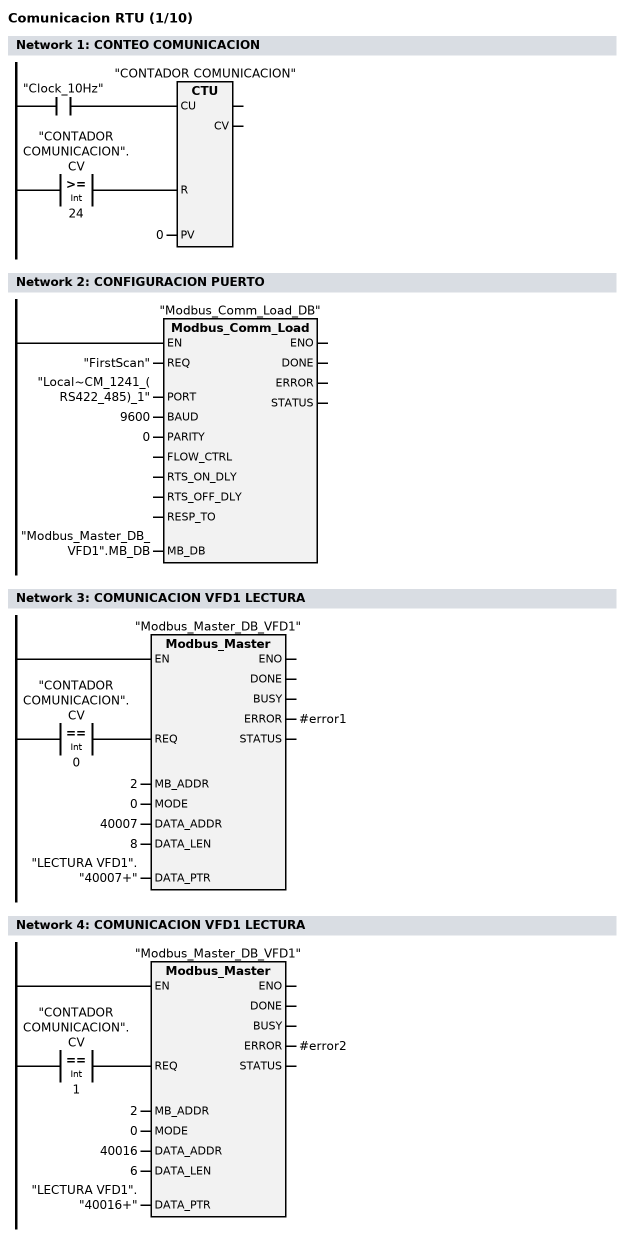
   "CONTADOR COMUNICACION".CTU(CU := "Clock_10Hz", R := "CONTADOR COMUNICACION".CV >= 24, PV := 0);
END_REGION

REGION Network 2: CONFIGURACION PUERTO
   "Modbus_Comm_Load_DB"(REQ := "FirstScan",   // Modbus_Comm_Load
                         PORT := "Local~CM_1241_(RS422_485)_1",
                         BAUD := 9600,
                         PARITY := 0,
                         MB_DB := "Modbus_Master_DB_VFD1".MB_DB);
END_REGION

REGION Network 3: COMUNICACION VFD1 LECTURA
   "Modbus_Master_DB_VFD1"(REQ := "CONTADOR COMUNICACION".CV = 0,   // Modbus_Master
                           MB_ADDR := 2,
                           MODE := 0,
                           DATA_ADDR := 40007,
                           DATA_LEN := 8,
                           DATA_PTR := "LECTURA VFD1"."40007+",
                           ERROR => #error1);
END_REGION

REGION Network 4: COMUNICACION VFD1 LECTURA
   "Modbus_Master_DB_VFD1"(REQ := "CONTADOR COMUNICACION".CV = 1,   // Modbus_Master
                           MB_ADDR := 2,
                           MODE := 0,
                           DATA_ADDR := 40016,
                           DATA_LEN := 6,
                           DATA_PTR := "LECTURA VFD1"."40016+",
                           ERROR => #error2);
END_REGION

REGION Network 5: COMUNICACION VFD2 LECTURA
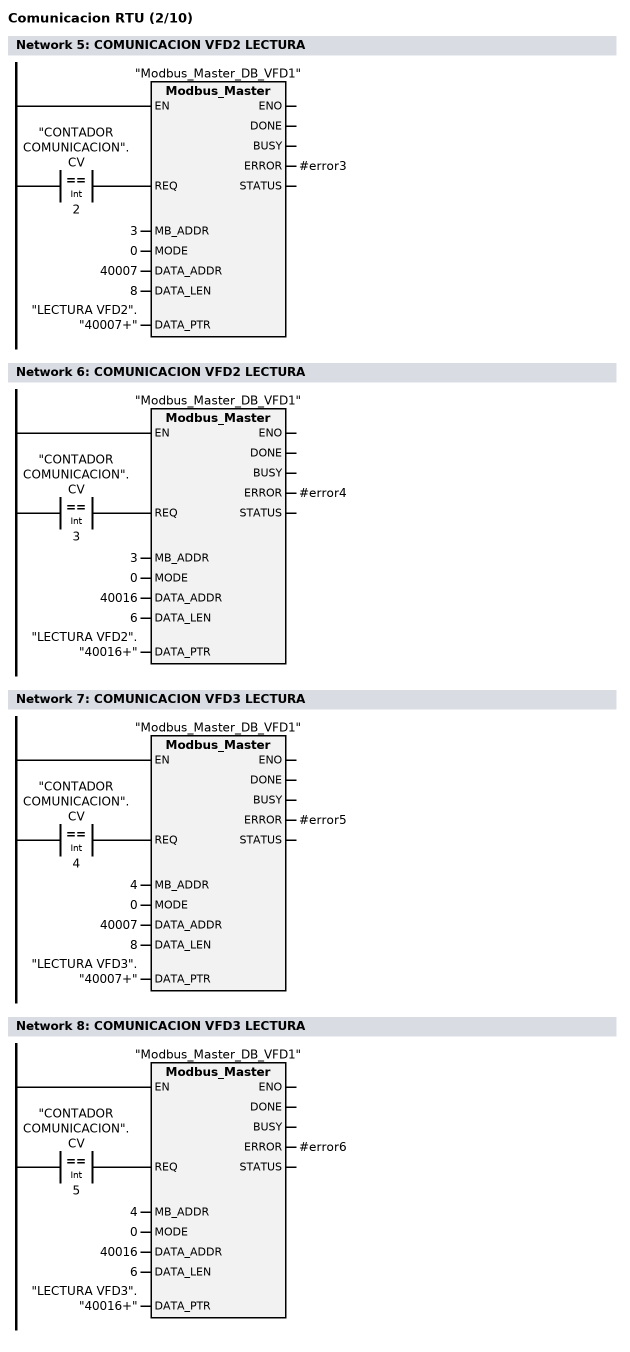
   "Modbus_Master_DB_VFD1"(REQ := "CONTADOR COMUNICACION".CV = 2,   // Modbus_Master
                           MB_ADDR := 3,
                           MODE := 0,
                           DATA_ADDR := 40007,
                           DATA_LEN := 8,
                           DATA_PTR := "LECTURA VFD2"."40007+",
                           ERROR => #error3);
END_REGION

REGION Network 6: COMUNICACION VFD2 LECTURA
   "Modbus_Master_DB_VFD1"(REQ := "CONTADOR COMUNICACION".CV = 3,   // Modbus_Master
                           MB_ADDR := 3,
                           MODE := 0,
                           DATA_ADDR := 40016,
                           DATA_LEN := 6,
                           DATA_PTR := "LECTURA VFD2"."40016+",
                           ERROR => #error4);
END_REGION

REGION Network 7: COMUNICACION VFD3 LECTURA
   "Modbus_Master_DB_VFD1"(REQ := "CONTADOR COMUNICACION".CV = 4,   // Modbus_Master
                           MB_ADDR := 4,
                           MODE := 0,
                           DATA_ADDR := 40007,
                           DATA_LEN := 8,
                           DATA_PTR := "LECTURA VFD3"."40007+",
                           ERROR => #error5);
END_REGION

REGION Network 8: COMUNICACION VFD3 LECTURA
   "Modbus_Master_DB_VFD1"(REQ := "CONTADOR COMUNICACION".CV = 5,   // Modbus_Master
                           MB_ADDR := 4,
                           MODE := 0,
                           DATA_ADDR := 40016,
                           DATA_LEN := 6,
                           DATA_PTR := "LECTURA VFD3"."40016+",
                           ERROR => #error6);
END_REGION

REGION Network 9: COMUNICACION VFD4 LECTURA
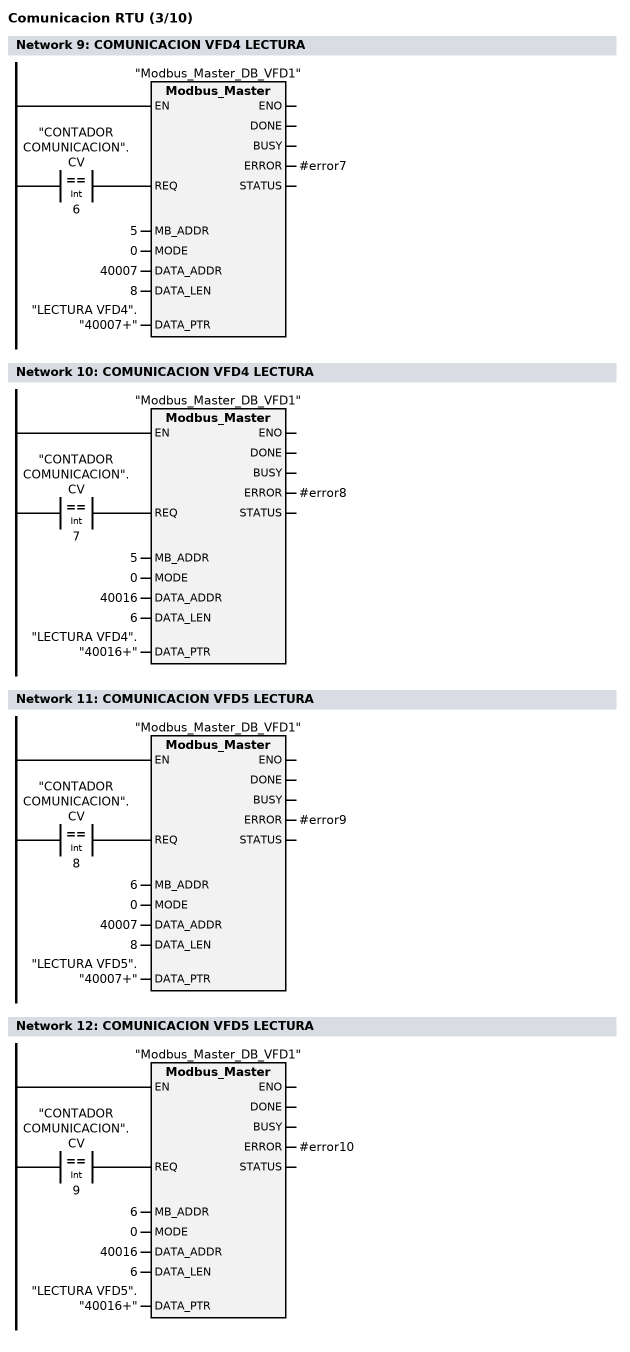
   "Modbus_Master_DB_VFD1"(REQ := "CONTADOR COMUNICACION".CV = 6,   // Modbus_Master
                           MB_ADDR := 5,
                           MODE := 0,
                           DATA_ADDR := 40007,
                           DATA_LEN := 8,
                           DATA_PTR := "LECTURA VFD4"."40007+",
                           ERROR => #error7);
END_REGION

REGION Network 10: COMUNICACION VFD4 LECTURA
   "Modbus_Master_DB_VFD1"(REQ := "CONTADOR COMUNICACION".CV = 7,   // Modbus_Master
                           MB_ADDR := 5,
                           MODE := 0,
                           DATA_ADDR := 40016,
                           DATA_LEN := 6,
                           DATA_PTR := "LECTURA VFD4"."40016+",
                           ERROR => #error8);
END_REGION

REGION Network 11: COMUNICACION VFD5 LECTURA
   "Modbus_Master_DB_VFD1"(REQ := "CONTADOR COMUNICACION".CV = 8,   // Modbus_Master
                           MB_ADDR := 6,
                           MODE := 0,
                           DATA_ADDR := 40007,
                           DATA_LEN := 8,
                           DATA_PTR := "LECTURA VFD5"."40007+",
                           ERROR => #error9);
END_REGION

REGION Network 12: COMUNICACION VFD5 LECTURA
   "Modbus_Master_DB_VFD1"(REQ := "CONTADOR COMUNICACION".CV = 9,   // Modbus_Master
                           MB_ADDR := 6,
                           MODE := 0,
                           DATA_ADDR := 40016,
                           DATA_LEN := 6,
                           DATA_PTR := "LECTURA VFD5"."40016+",
                           ERROR => #error10);
END_REGION

REGION Network 13: COMUNICACION VFD6 LECTURA
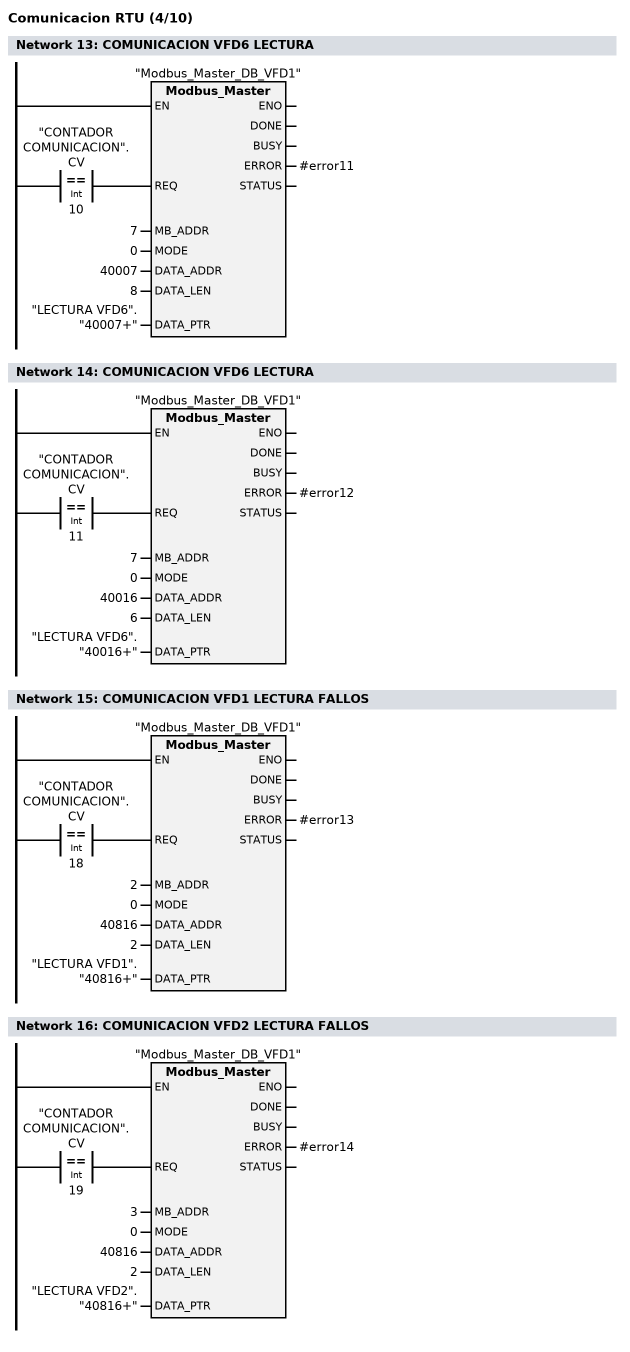
   "Modbus_Master_DB_VFD1"(REQ := "CONTADOR COMUNICACION".CV = 10,   // Modbus_Master
                           MB_ADDR := 7,
                           MODE := 0,
                           DATA_ADDR := 40007,
                           DATA_LEN := 8,
                           DATA_PTR := "LECTURA VFD6"."40007+",
                           ERROR => #error11);
END_REGION

REGION Network 14: COMUNICACION VFD6 LECTURA
   "Modbus_Master_DB_VFD1"(REQ := "CONTADOR COMUNICACION".CV = 11,   // Modbus_Master
                           MB_ADDR := 7,
                           MODE := 0,
                           DATA_ADDR := 40016,
                           DATA_LEN := 6,
                           DATA_PTR := "LECTURA VFD6"."40016+",
                           ERROR => #error12);
END_REGION

REGION Network 15: COMUNICACION VFD1 LECTURA FALLOS
   "Modbus_Master_DB_VFD1"(REQ := "CONTADOR COMUNICACION".CV = 18,   // Modbus_Master
                           MB_ADDR := 2,
                           MODE := 0,
                           DATA_ADDR := 40816,
                           DATA_LEN := 2,
                           DATA_PTR := "LECTURA VFD1"."40816+",
                           ERROR => #error13);
END_REGION

REGION Network 16: COMUNICACION VFD2 LECTURA FALLOS
   "Modbus_Master_DB_VFD1"(REQ := "CONTADOR COMUNICACION".CV = 19,   // Modbus_Master
                           MB_ADDR := 3,
                           MODE := 0,
                           DATA_ADDR := 40816,
                           DATA_LEN := 2,
                           DATA_PTR := "LECTURA VFD2"."40816+",
                           ERROR => #error14);
END_REGION

REGION Network 17: COMUNICACION VFD3 LECTURA FALLOS
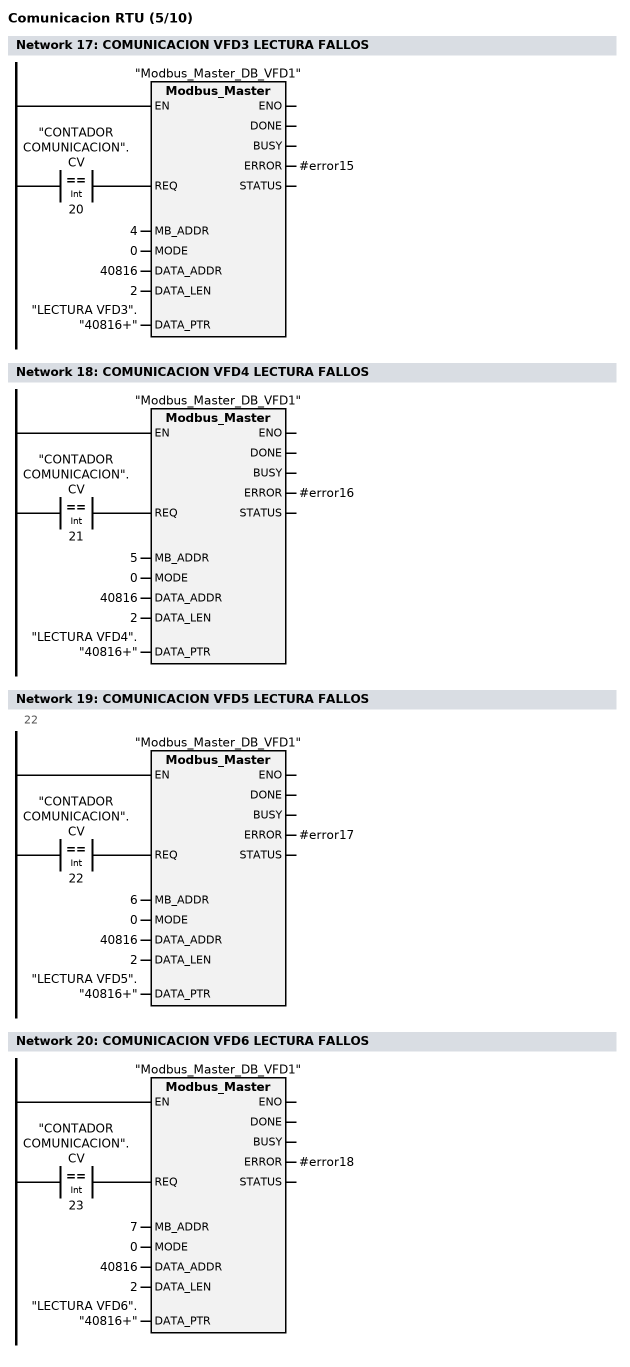
   "Modbus_Master_DB_VFD1"(REQ := "CONTADOR COMUNICACION".CV = 20,   // Modbus_Master
                           MB_ADDR := 4,
                           MODE := 0,
                           DATA_ADDR := 40816,
                           DATA_LEN := 2,
                           DATA_PTR := "LECTURA VFD3"."40816+",
                           ERROR => #error15);
END_REGION

REGION Network 18: COMUNICACION VFD4 LECTURA FALLOS
   "Modbus_Master_DB_VFD1"(REQ := "CONTADOR COMUNICACION".CV = 21,   // Modbus_Master
                           MB_ADDR := 5,
                           MODE := 0,
                           DATA_ADDR := 40816,
                           DATA_LEN := 2,
                           DATA_PTR := "LECTURA VFD4"."40816+",
                           ERROR => #error16);
END_REGION

REGION Network 19: COMUNICACION VFD5 LECTURA FALLOS
   // 22
   "Modbus_Master_DB_VFD1"(REQ := "CONTADOR COMUNICACION".CV = 22,   // Modbus_Master
                           MB_ADDR := 6,
                           MODE := 0,
                           DATA_ADDR := 40816,
                           DATA_LEN := 2,
                           DATA_PTR := "LECTURA VFD5"."40816+",
                           ERROR => #error17);
END_REGION

REGION Network 20: COMUNICACION VFD6 LECTURA FALLOS
   "Modbus_Master_DB_VFD1"(REQ := "CONTADOR COMUNICACION".CV = 23,   // Modbus_Master
                           MB_ADDR := 7,
                           MODE := 0,
                           DATA_ADDR := 40816,
                           DATA_LEN := 2,
                           DATA_PTR := "LECTURA VFD6"."40816+",
                           ERROR => #error18);
END_REGION

REGION Network 21: COMUNICACION VFD1 ESCRITURA
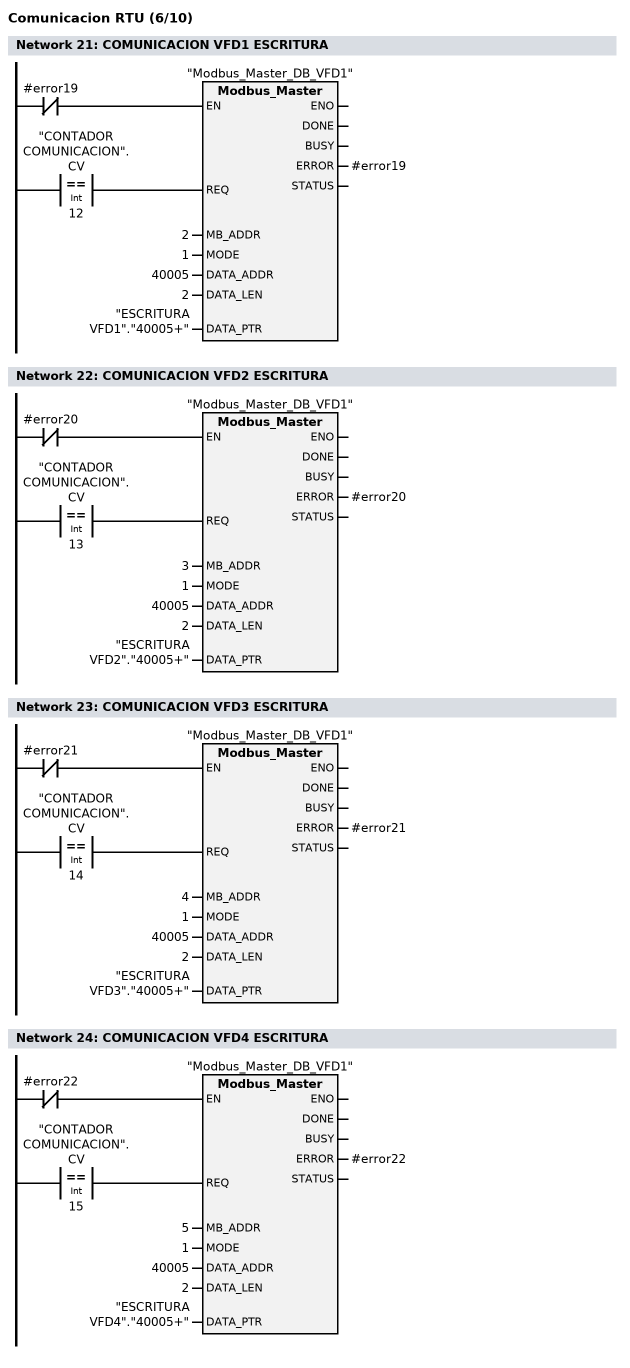
   IF NOT #error19 THEN
       "Modbus_Master_DB_VFD1"(REQ := "CONTADOR COMUNICACION".CV = 12,   // Modbus_Master
                               MB_ADDR := 2,
                               MODE := 1,
                               DATA_ADDR := 40005,
                               DATA_LEN := 2,
                               DATA_PTR := "ESCRITURA VFD1"."40005+",
                               ERROR => #error19);
   END_IF;
END_REGION

REGION Network 22: COMUNICACION VFD2 ESCRITURA
   IF NOT #error20 THEN
       "Modbus_Master_DB_VFD1"(REQ := "CONTADOR COMUNICACION".CV = 13,   // Modbus_Master
                               MB_ADDR := 3,
                               MODE := 1,
                               DATA_ADDR := 40005,
                               DATA_LEN := 2,
                               DATA_PTR := "ESCRITURA VFD2"."40005+",
                               ERROR => #error20);
   END_IF;
END_REGION

REGION Network 23: COMUNICACION VFD3 ESCRITURA
   IF NOT #error21 THEN
       "Modbus_Master_DB_VFD1"(REQ := "CONTADOR COMUNICACION".CV = 14,   // Modbus_Master
                               MB_ADDR := 4,
                               MODE := 1,
                               DATA_ADDR := 40005,
                               DATA_LEN := 2,
                               DATA_PTR := "ESCRITURA VFD3"."40005+",
                               ERROR => #error21);
   END_IF;
END_REGION

REGION Network 24: COMUNICACION VFD4 ESCRITURA
   IF NOT #error22 THEN
       "Modbus_Master_DB_VFD1"(REQ := "CONTADOR COMUNICACION".CV = 15,   // Modbus_Master
                               MB_ADDR := 5,
                               MODE := 1,
                               DATA_ADDR := 40005,
                               DATA_LEN := 2,
                               DATA_PTR := "ESCRITURA VFD4"."40005+",
                               ERROR => #error22);
   END_IF;
END_REGION

REGION Network 25: COMUNICACION VFD5 ESCRITURA
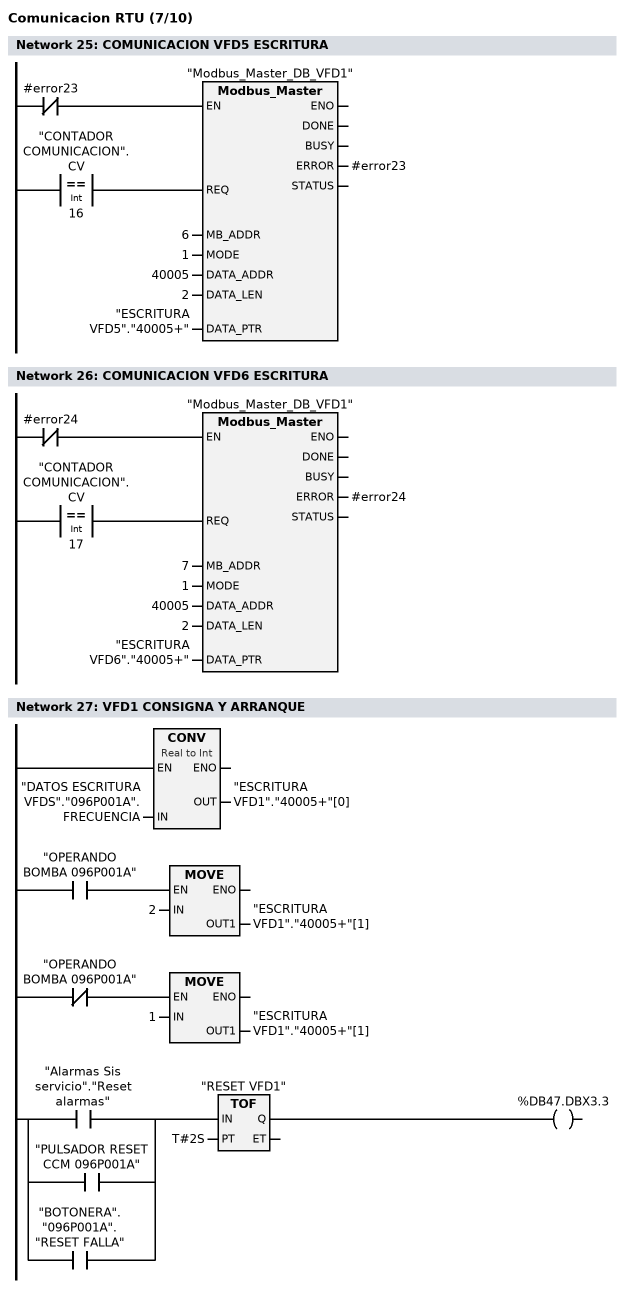
   IF NOT #error23 THEN
       "Modbus_Master_DB_VFD1"(REQ := "CONTADOR COMUNICACION".CV = 16,   // Modbus_Master
                               MB_ADDR := 6,
                               MODE := 1,
                               DATA_ADDR := 40005,
                               DATA_LEN := 2,
                               DATA_PTR := "ESCRITURA VFD5"."40005+",
                               ERROR => #error23);
   END_IF;
END_REGION

REGION Network 26: COMUNICACION VFD6 ESCRITURA
   IF NOT #error24 THEN
       "Modbus_Master_DB_VFD1"(REQ := "CONTADOR COMUNICACION".CV = 17,   // Modbus_Master
                               MB_ADDR := 7,
                               MODE := 1,
                               DATA_ADDR := 40005,
                               DATA_LEN := 2,
                               DATA_PTR := "ESCRITURA VFD6"."40005+",
                               ERROR => #error24);
   END_IF;
END_REGION

REGION Network 27: VFD1 CONSIGNA Y ARRANQUE
   "ESCRITURA VFD1"."40005+"[0] := REAL_TO_INT("DATOS ESCRITURA VFDS"."096P001A".FRECUENCIA);
   IF "OPERANDO BOMBA 096P001A" THEN "ESCRITURA VFD1"."40005+"[1] := 2; END_IF;
   IF NOT "OPERANDO BOMBA 096P001A" THEN "ESCRITURA VFD1"."40005+"[1] := 1; END_IF;
   "RESET VFD1".TOF(IN := "Alarmas Sis servicio"."Reset alarmas" OR "PULSADOR RESET CCM 096P001A" OR "BOTONERA"."096P001A"."RESET FALLA",
                    PT := T#2S);
   %DB47.DBX3.3 := "RESET VFD1".Q;
END_REGION

REGION Network 28: VFD2 CONSIGNA Y ARRANQUE
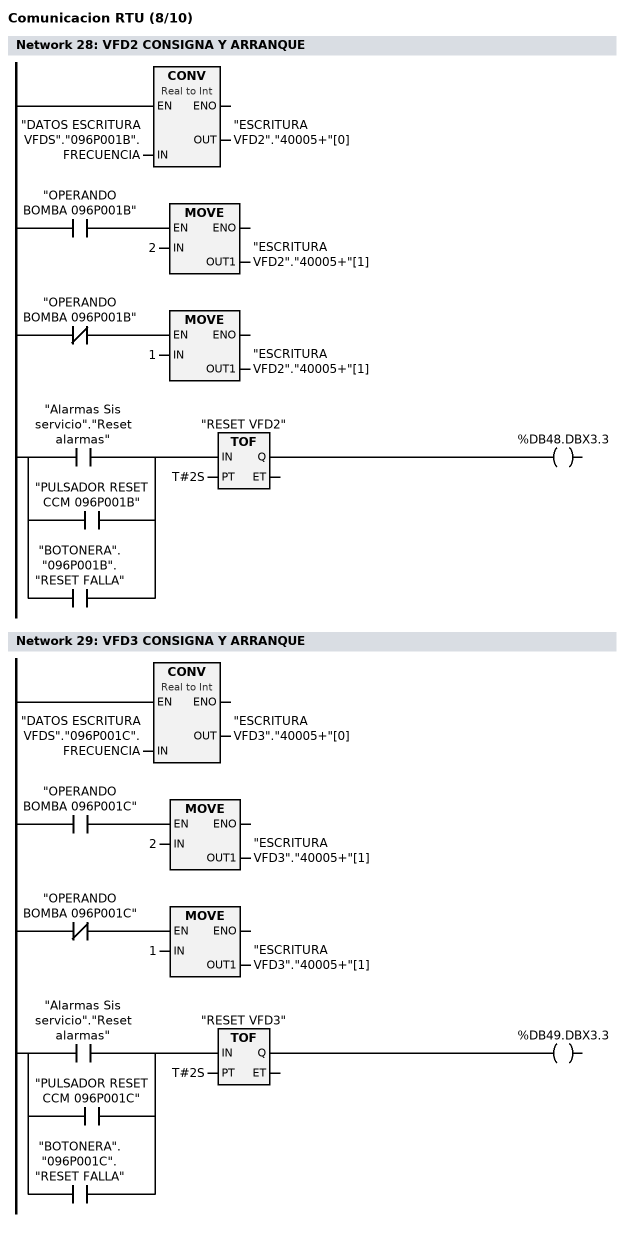
   "ESCRITURA VFD2"."40005+"[0] := REAL_TO_INT("DATOS ESCRITURA VFDS"."096P001B".FRECUENCIA);
   IF "OPERANDO BOMBA 096P001B" THEN "ESCRITURA VFD2"."40005+"[1] := 2; END_IF;
   IF NOT "OPERANDO BOMBA 096P001B" THEN "ESCRITURA VFD2"."40005+"[1] := 1; END_IF;
   "RESET VFD2".TOF(IN := "Alarmas Sis servicio"."Reset alarmas" OR "PULSADOR RESET CCM 096P001B" OR "BOTONERA"."096P001B"."RESET FALLA",
                    PT := T#2S);
   %DB48.DBX3.3 := "RESET VFD2".Q;
END_REGION

REGION Network 29: VFD3 CONSIGNA Y ARRANQUE
   "ESCRITURA VFD3"."40005+"[0] := REAL_TO_INT("DATOS ESCRITURA VFDS"."096P001C".FRECUENCIA);
   IF "OPERANDO BOMBA 096P001C" THEN "ESCRITURA VFD3"."40005+"[1] := 2; END_IF;
   IF NOT "OPERANDO BOMBA 096P001C" THEN "ESCRITURA VFD3"."40005+"[1] := 1; END_IF;
   "RESET VFD3".TOF(IN := "Alarmas Sis servicio"."Reset alarmas" OR "PULSADOR RESET CCM 096P001C" OR "BOTONERA"."096P001C"."RESET FALLA",
                    PT := T#2S);
   %DB49.DBX3.3 := "RESET VFD3".Q;
END_REGION

REGION Network 30: VFD4 CONSIGNA Y ARRANQUE
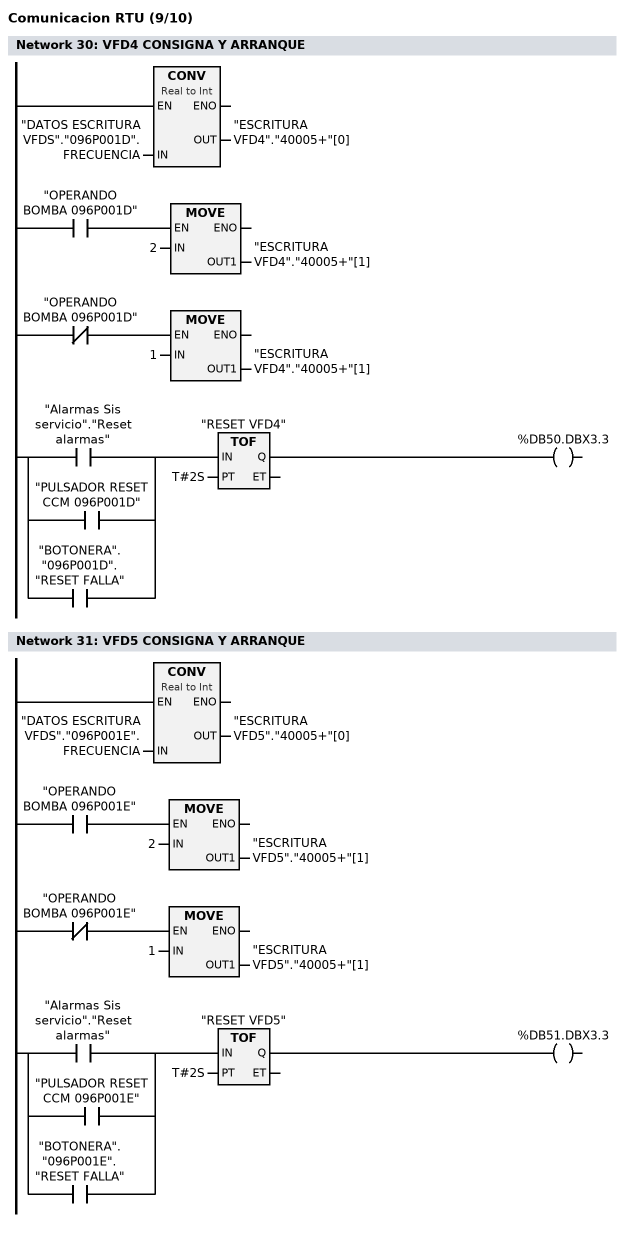
   "ESCRITURA VFD4"."40005+"[0] := REAL_TO_INT("DATOS ESCRITURA VFDS"."096P001D".FRECUENCIA);
   IF "OPERANDO BOMBA 096P001D" THEN "ESCRITURA VFD4"."40005+"[1] := 2; END_IF;
   IF NOT "OPERANDO BOMBA 096P001D" THEN "ESCRITURA VFD4"."40005+"[1] := 1; END_IF;
   "RESET VFD4".TOF(IN := "Alarmas Sis servicio"."Reset alarmas" OR "PULSADOR RESET CCM 096P001D" OR "BOTONERA"."096P001D"."RESET FALLA",
                    PT := T#2S);
   %DB50.DBX3.3 := "RESET VFD4".Q;
END_REGION

REGION Network 31: VFD5 CONSIGNA Y ARRANQUE
   "ESCRITURA VFD5"."40005+"[0] := REAL_TO_INT("DATOS ESCRITURA VFDS"."096P001E".FRECUENCIA);
   IF "OPERANDO BOMBA 096P001E" THEN "ESCRITURA VFD5"."40005+"[1] := 2; END_IF;
   IF NOT "OPERANDO BOMBA 096P001E" THEN "ESCRITURA VFD5"."40005+"[1] := 1; END_IF;
   "RESET VFD5".TOF(IN := "Alarmas Sis servicio"."Reset alarmas" OR "PULSADOR RESET CCM 096P001E" OR "BOTONERA"."096P001E"."RESET FALLA",
                    PT := T#2S);
   %DB51.DBX3.3 := "RESET VFD5".Q;
END_REGION

REGION Network 32: VFD6 CONSIGNA Y ARRANQUE
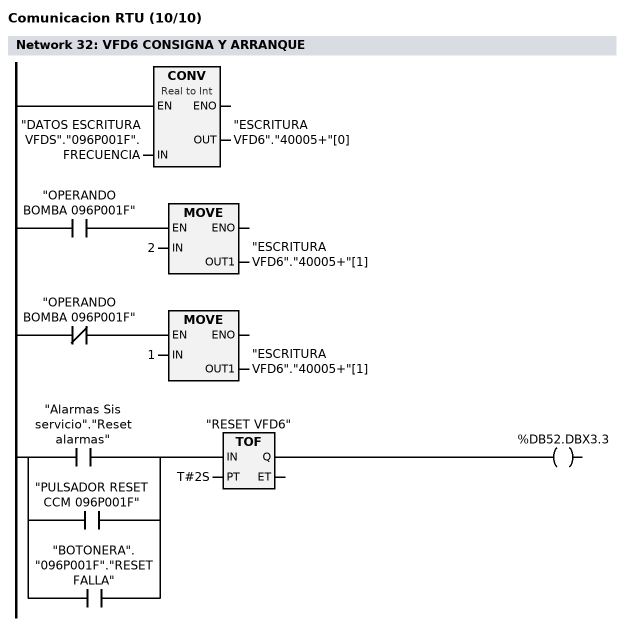
   "ESCRITURA VFD6"."40005+"[0] := REAL_TO_INT("DATOS ESCRITURA VFDS"."096P001F".FRECUENCIA);
   IF "OPERANDO BOMBA 096P001F" THEN "ESCRITURA VFD6"."40005+"[1] := 2; END_IF;
   IF NOT "OPERANDO BOMBA 096P001F" THEN "ESCRITURA VFD6"."40005+"[1] := 1; END_IF;
   "RESET VFD6".TOF(IN := "Alarmas Sis servicio"."Reset alarmas" OR "PULSADOR RESET CCM 096P001F" OR "BOTONERA"."096P001F"."RESET FALLA",
                    PT := T#2S);
   %DB52.DBX3.3 := "RESET VFD6".Q;
END_REGION
END_FUNCTION

FUNCTION "DATOS HMI" : Void   // FC6, LAD
{ S7_Optimized_Access := 'TRUE' }
VERSION : 0.1
BEGIN

REGION Network 1: VFD1
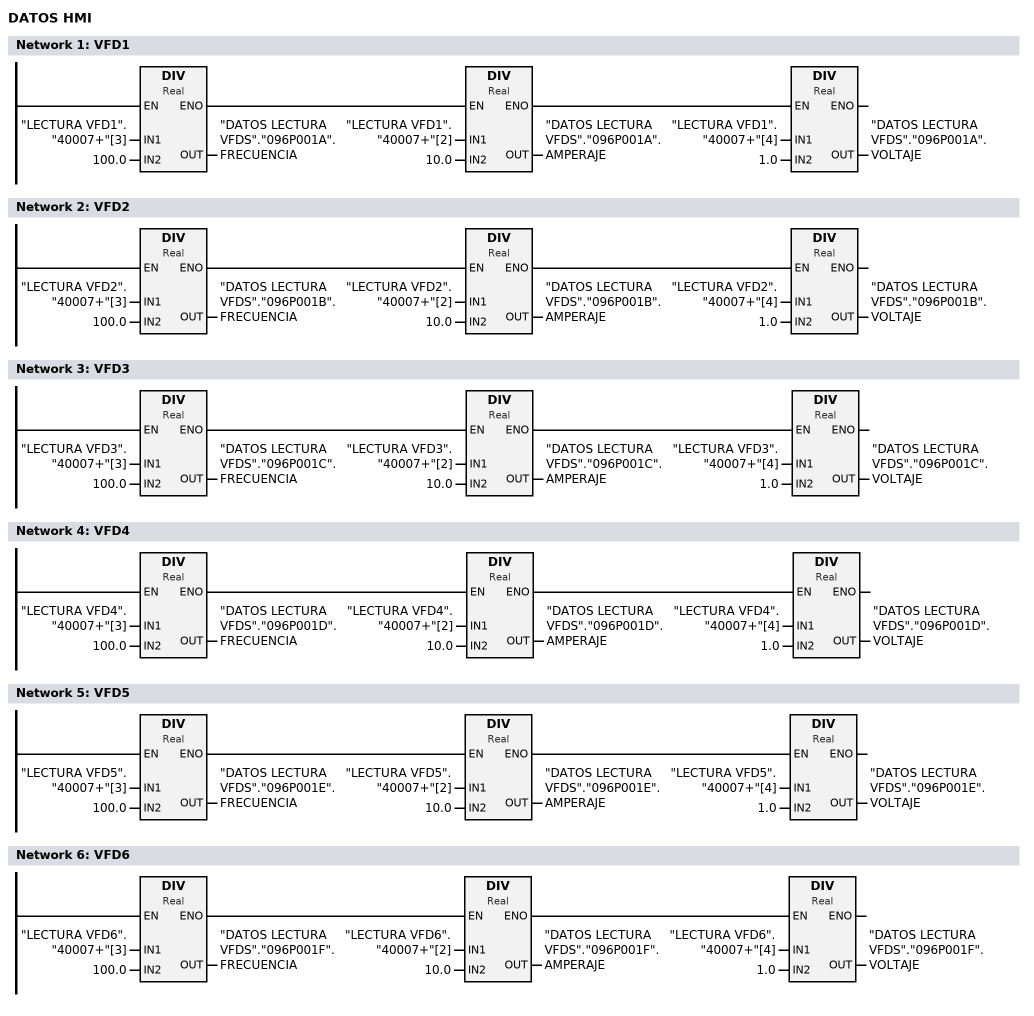
   RUNG wire#powerrail
      { S7_Templates := "SrcType := Real" } Div(in1 := "LECTURA VFD1"."40007+"[3], in2 := 100.0, out => "DATOS LECTURA VFDS"."096P001A".FRECUENCIA)
      { S7_Templates := "SrcType := Real" } Div(in1 := "LECTURA VFD1"."40007+"[2], in2 := 10.0, out => "DATOS LECTURA VFDS"."096P001A".AMPERAJE)
      { S7_Templates := "SrcType := Real" } Div(in1 := "LECTURA VFD1"."40007+"[4], in2 := 1.0, out => "DATOS LECTURA VFDS"."096P001A".VOLTAJE)
   END_RUNG
   // the same network as SCL:
   "DATOS LECTURA VFDS"."096P001A".FRECUENCIA := "LECTURA VFD1"."40007+"[3] / 100.0;
   "DATOS LECTURA VFDS"."096P001A".AMPERAJE := "LECTURA VFD1"."40007+"[2] / 10.0;
   "DATOS LECTURA VFDS"."096P001A".VOLTAJE := "LECTURA VFD1"."40007+"[4] / 1.0;
END_REGION

REGION Network 2: VFD2
   RUNG wire#powerrail
      { S7_Templates := "SrcType := Real" } Div(in1 := "LECTURA VFD2"."40007+"[3], in2 := 100.0, out => "DATOS LECTURA VFDS"."096P001B".FRECUENCIA)
      { S7_Templates := "SrcType := Real" } Div(in1 := "LECTURA VFD2"."40007+"[2], in2 := 10.0, out => "DATOS LECTURA VFDS"."096P001B".AMPERAJE)
      { S7_Templates := "SrcType := Real" } Div(in1 := "LECTURA VFD2"."40007+"[4], in2 := 1.0, out => "DATOS LECTURA VFDS"."096P001B".VOLTAJE)
   END_RUNG
   // the same network as SCL:
   "DATOS LECTURA VFDS"."096P001B".FRECUENCIA := "LECTURA VFD2"."40007+"[3] / 100.0;
   "DATOS LECTURA VFDS"."096P001B".AMPERAJE := "LECTURA VFD2"."40007+"[2] / 10.0;
   "DATOS LECTURA VFDS"."096P001B".VOLTAJE := "LECTURA VFD2"."40007+"[4] / 1.0;
END_REGION

REGION Network 3: VFD3
   RUNG wire#powerrail
      { S7_Templates := "SrcType := Real" } Div(in1 := "LECTURA VFD3"."40007+"[3], in2 := 100.0, out => "DATOS LECTURA VFDS"."096P001C".FRECUENCIA)
      { S7_Templates := "SrcType := Real" } Div(in1 := "LECTURA VFD3"."40007+"[2], in2 := 10.0, out => "DATOS LECTURA VFDS"."096P001C".AMPERAJE)
      { S7_Templates := "SrcType := Real" } Div(in1 := "LECTURA VFD3"."40007+"[4], in2 := 1.0, out => "DATOS LECTURA VFDS"."096P001C".VOLTAJE)
   END_RUNG
   // the same network as SCL:
   "DATOS LECTURA VFDS"."096P001C".FRECUENCIA := "LECTURA VFD3"."40007+"[3] / 100.0;
   "DATOS LECTURA VFDS"."096P001C".AMPERAJE := "LECTURA VFD3"."40007+"[2] / 10.0;
   "DATOS LECTURA VFDS"."096P001C".VOLTAJE := "LECTURA VFD3"."40007+"[4] / 1.0;
END_REGION

REGION Network 4: VFD4
   RUNG wire#powerrail
      { S7_Templates := "SrcType := Real" } Div(in1 := "LECTURA VFD4"."40007+"[3], in2 := 100.0, out => "DATOS LECTURA VFDS"."096P001D".FRECUENCIA)
      { S7_Templates := "SrcType := Real" } Div(in1 := "LECTURA VFD4"."40007+"[2], in2 := 10.0, out => "DATOS LECTURA VFDS"."096P001D".AMPERAJE)
      { S7_Templates := "SrcType := Real" } Div(in1 := "LECTURA VFD4"."40007+"[4], in2 := 1.0, out => "DATOS LECTURA VFDS"."096P001D".VOLTAJE)
   END_RUNG
   // the same network as SCL:
   "DATOS LECTURA VFDS"."096P001D".FRECUENCIA := "LECTURA VFD4"."40007+"[3] / 100.0;
   "DATOS LECTURA VFDS"."096P001D".AMPERAJE := "LECTURA VFD4"."40007+"[2] / 10.0;
   "DATOS LECTURA VFDS"."096P001D".VOLTAJE := "LECTURA VFD4"."40007+"[4] / 1.0;
END_REGION

REGION Network 5: VFD5
   RUNG wire#powerrail
      { S7_Templates := "SrcType := Real" } Div(in1 := "LECTURA VFD5"."40007+"[3], in2 := 100.0, out => "DATOS LECTURA VFDS"."096P001E".FRECUENCIA)
      { S7_Templates := "SrcType := Real" } Div(in1 := "LECTURA VFD5"."40007+"[2], in2 := 10.0, out => "DATOS LECTURA VFDS"."096P001E".AMPERAJE)
      { S7_Templates := "SrcType := Real" } Div(in1 := "LECTURA VFD5"."40007+"[4], in2 := 1.0, out => "DATOS LECTURA VFDS"."096P001E".VOLTAJE)
   END_RUNG
   // the same network as SCL:
   "DATOS LECTURA VFDS"."096P001E".FRECUENCIA := "LECTURA VFD5"."40007+"[3] / 100.0;
   "DATOS LECTURA VFDS"."096P001E".AMPERAJE := "LECTURA VFD5"."40007+"[2] / 10.0;
   "DATOS LECTURA VFDS"."096P001E".VOLTAJE := "LECTURA VFD5"."40007+"[4] / 1.0;
END_REGION

REGION Network 6: VFD6
   RUNG wire#powerrail
      { S7_Templates := "SrcType := Real" } Div(in1 := "LECTURA VFD6"."40007+"[3], in2 := 100.0, out => "DATOS LECTURA VFDS"."096P001F".FRECUENCIA)
      { S7_Templates := "SrcType := Real" } Div(in1 := "LECTURA VFD6"."40007+"[2], in2 := 10.0, out => "DATOS LECTURA VFDS"."096P001F".AMPERAJE)
      { S7_Templates := "SrcType := Real" } Div(in1 := "LECTURA VFD6"."40007+"[4], in2 := 1.0, out => "DATOS LECTURA VFDS"."096P001F".VOLTAJE)
   END_RUNG
   // the same network as SCL:
   "DATOS LECTURA VFDS"."096P001F".FRECUENCIA := "LECTURA VFD6"."40007+"[3] / 100.0;
   "DATOS LECTURA VFDS"."096P001F".AMPERAJE := "LECTURA VFD6"."40007+"[2] / 10.0;
   "DATOS LECTURA VFDS"."096P001F".VOLTAJE := "LECTURA VFD6"."40007+"[4] / 1.0;
END_REGION
END_FUNCTION

FUNCTION "COMUNICACION MODBUS TCP" : Void   // FC7, LAD
{ S7_Optimized_Access := 'TRUE' }
VERSION : 0.1
   VAR_TEMP
      "REAL 1" : Real;
      "REAL 2" : Real;
      "REAL 3" : Real;
      "REAL 4" : Real;
      "REAL 5" : Real;
      "REAL 6" : Real;
      "REAL 7" : Real;
      "REAL 8" : Real;
      "REAL 9" : Real;
      "REAL 10" : Real;
      "REAL 11" : Real;
      "REAL 12" : Real;
      "REAL 13" : Real;
      "REAL 14" : Real;
      "REAL 15" : Real;
      "REAL 16" : Real;
      "REAL 17" : Real;
      "REAL 18" : Real;
      "REAL 19" : Real;
      "REAL 20" : Real;
      "REAL 21" : Real;
      "REAL 22" : Real;
      "REAL 23" : Real;
      "REAL 24" : Real;
      "REAL 25" : Real;
      "REAL 26" : Real;
      "REAL 27" : Real;
      "REAL 28" : Real;
      "REAL 29" : Real;
      "REAL 30" : Real;
   END_VAR
   VAR_TEMP   // added for the SCL form of the ladder/FBD networks
      _w1 : Bool;
      _w2 : Bool;
      _w3 : Bool;
   END_VAR
BEGIN

REGION Network 1: CONFIGURACION MODBUS TCP
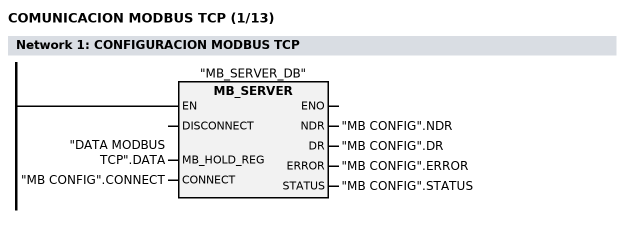
   "MB_SERVER_DB"(MB_HOLD_REG := "DATA MODBUS TCP".DATA,   // MB_SERVER
                  CONNECT := "MB CONFIG".CONNECT,
                  NDR => "MB CONFIG".NDR,
                  DR => "MB CONFIG".DR,
                  ERROR => "MB CONFIG".ERROR,
                  STATUS => "MB CONFIG".STATUS);
END_REGION

REGION Network 2: ENTRADAS DIGITALES
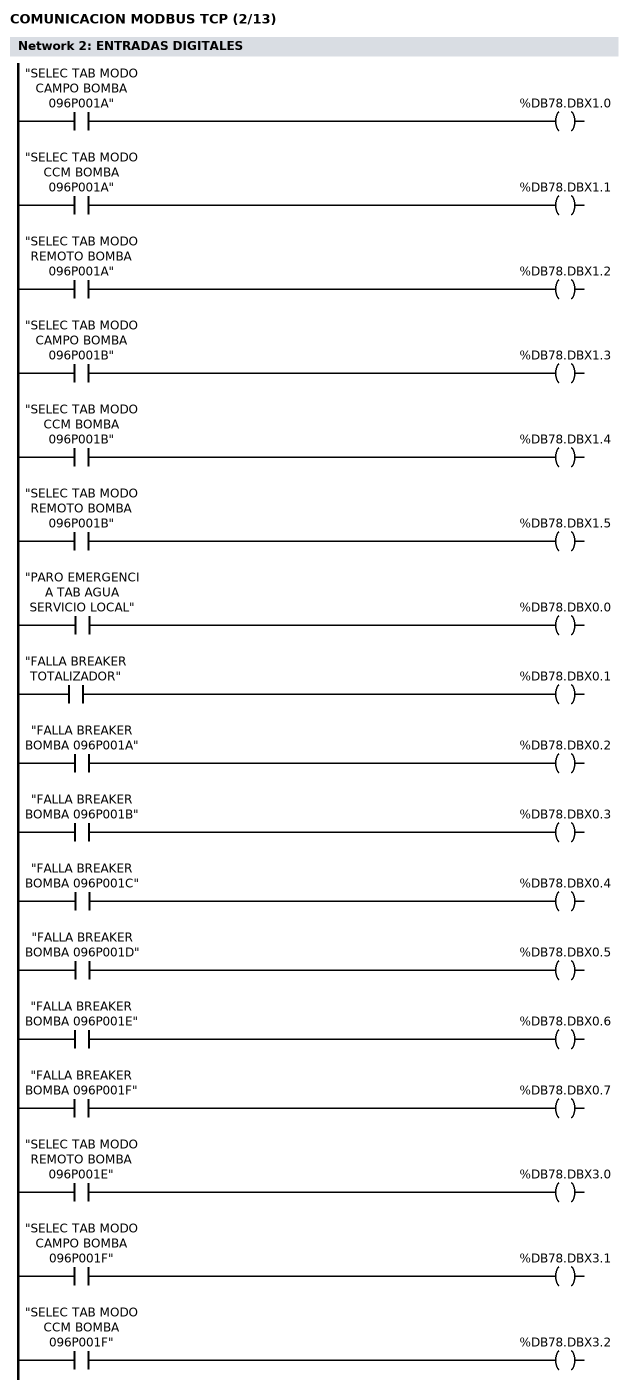
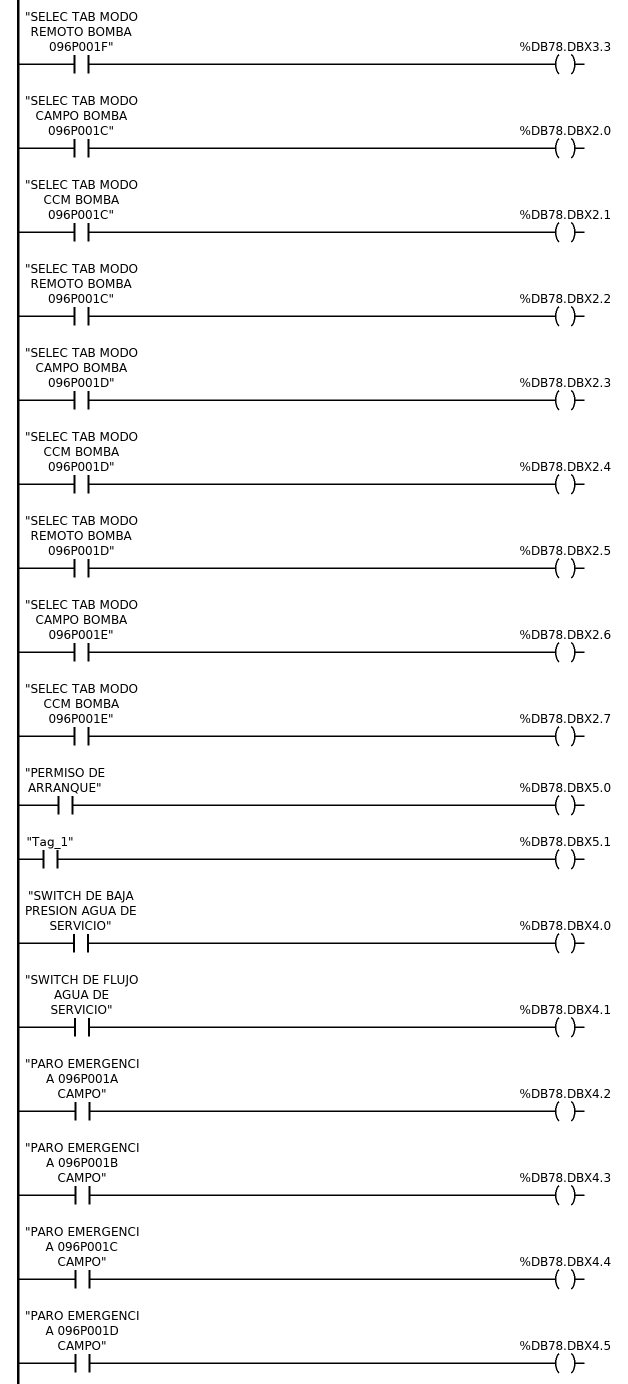
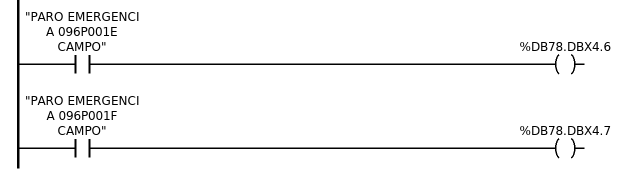
   RUNG wire#powerrail
      Contact( "SELEC TAB MODO CAMPO BOMBA 096P001A" )
      Coil( %DB78.DBX1.0 )
   END_RUNG
   RUNG wire#powerrail
      Contact( "SELEC TAB MODO CCM BOMBA 096P001A" )
      Coil( %DB78.DBX1.1 )
   END_RUNG
   RUNG wire#powerrail
      Contact( "SELEC TAB MODO REMOTO BOMBA 096P001A" )
      Coil( %DB78.DBX1.2 )
   END_RUNG
   RUNG wire#powerrail
      Contact( "SELEC TAB MODO CAMPO BOMBA 096P001B" )
      Coil( %DB78.DBX1.3 )
   END_RUNG
   RUNG wire#powerrail
      Contact( "SELEC TAB MODO CCM BOMBA 096P001B" )
      Coil( %DB78.DBX1.4 )
   END_RUNG
   RUNG wire#powerrail
      Contact( "SELEC TAB MODO REMOTO BOMBA 096P001B" )
      Coil( %DB78.DBX1.5 )
   END_RUNG
   RUNG wire#powerrail
      Contact( "PARO EMERGENCIA TAB AGUA SERVICIO LOCAL" )
      Coil( %DB78.DBX0.0 )
   END_RUNG
   RUNG wire#powerrail
      Contact( "FALLA BREAKER TOTALIZADOR" )
      Coil( %DB78.DBX0.1 )
   END_RUNG
   RUNG wire#powerrail
      Contact( "FALLA BREAKER BOMBA 096P001A" )
      Coil( %DB78.DBX0.2 )
   END_RUNG
   RUNG wire#powerrail
      Contact( "FALLA BREAKER BOMBA 096P001B" )
      Coil( %DB78.DBX0.3 )
   END_RUNG
   RUNG wire#powerrail
      Contact( "FALLA BREAKER BOMBA 096P001C" )
      Coil( %DB78.DBX0.4 )
   END_RUNG
   RUNG wire#powerrail
      Contact( "FALLA BREAKER BOMBA 096P001D" )
      Coil( %DB78.DBX0.5 )
   END_RUNG
   RUNG wire#powerrail
      Contact( "FALLA BREAKER BOMBA 096P001E" )
      Coil( %DB78.DBX0.6 )
   END_RUNG
   RUNG wire#powerrail
      Contact( "FALLA BREAKER BOMBA 096P001F" )
      Coil( %DB78.DBX0.7 )
   END_RUNG
   RUNG wire#powerrail
      Contact( "SELEC TAB MODO REMOTO BOMBA 096P001E" )
      Coil( %DB78.DBX3.0 )
   END_RUNG
   RUNG wire#powerrail
      Contact( "SELEC TAB MODO CAMPO BOMBA 096P001F" )
      Coil( %DB78.DBX3.1 )
   END_RUNG
   RUNG wire#powerrail
      Contact( "SELEC TAB MODO CCM BOMBA 096P001F" )
      Coil( %DB78.DBX3.2 )
   END_RUNG
   RUNG wire#powerrail
      Contact( "SELEC TAB MODO REMOTO BOMBA 096P001F" )
      Coil( %DB78.DBX3.3 )
   END_RUNG
   RUNG wire#powerrail
      Contact( "SELEC TAB MODO CAMPO BOMBA 096P001C" )
      Coil( %DB78.DBX2.0 )
   END_RUNG
   RUNG wire#powerrail
      Contact( "SELEC TAB MODO CCM BOMBA 096P001C" )
      Coil( %DB78.DBX2.1 )
   END_RUNG
   RUNG wire#powerrail
      Contact( "SELEC TAB MODO REMOTO BOMBA 096P001C" )
      Coil( %DB78.DBX2.2 )
   END_RUNG
   RUNG wire#powerrail
      Contact( "SELEC TAB MODO CAMPO BOMBA 096P001D" )
      Coil( %DB78.DBX2.3 )
   END_RUNG
   RUNG wire#powerrail
      Contact( "SELEC TAB MODO CCM BOMBA 096P001D" )
      Coil( %DB78.DBX2.4 )
   END_RUNG
   RUNG wire#powerrail
      Contact( "SELEC TAB MODO REMOTO BOMBA 096P001D" )
      Coil( %DB78.DBX2.5 )
   END_RUNG
   RUNG wire#powerrail
      Contact( "SELEC TAB MODO CAMPO BOMBA 096P001E" )
      Coil( %DB78.DBX2.6 )
   END_RUNG
   RUNG wire#powerrail
      Contact( "SELEC TAB MODO CCM BOMBA 096P001E" )
      Coil( %DB78.DBX2.7 )
   END_RUNG
   RUNG wire#powerrail
      Contact( "PERMISO DE ARRANQUE" )
      Coil( %DB78.DBX5.0 )
   END_RUNG
   RUNG wire#powerrail
      Contact( "Tag_1" )
      Coil( %DB78.DBX5.1 )
   END_RUNG
   RUNG wire#powerrail
      Contact( "SWITCH DE BAJA PRESION AGUA DE SERVICIO" )
      Coil( %DB78.DBX4.0 )
   END_RUNG
   RUNG wire#powerrail
      Contact( "SWITCH DE FLUJO AGUA DE SERVICIO" )
      Coil( %DB78.DBX4.1 )
   END_RUNG
   RUNG wire#powerrail
      Contact( "PARO EMERGENCIA 096P001A CAMPO" )
      Coil( %DB78.DBX4.2 )
   END_RUNG
   RUNG wire#powerrail
      Contact( "PARO EMERGENCIA 096P001B CAMPO" )
      Coil( %DB78.DBX4.3 )
   END_RUNG
   RUNG wire#powerrail
      Contact( "PARO EMERGENCIA 096P001C CAMPO" )
      Coil( %DB78.DBX4.4 )
   END_RUNG
   RUNG wire#powerrail
      Contact( "PARO EMERGENCIA 096P001D CAMPO" )
      Coil( %DB78.DBX4.5 )
   END_RUNG
   RUNG wire#powerrail
      Contact( "PARO EMERGENCIA 096P001E CAMPO" )
      Coil( %DB78.DBX4.6 )
   END_RUNG
   RUNG wire#powerrail
      Contact( "PARO EMERGENCIA 096P001F CAMPO" )
      Coil( %DB78.DBX4.7 )
   END_RUNG
   // the same network as SCL:
   %DB78.DBX1.0 := "SELEC TAB MODO CAMPO BOMBA 096P001A";
   %DB78.DBX1.1 := "SELEC TAB MODO CCM BOMBA 096P001A";
   %DB78.DBX1.2 := "SELEC TAB MODO REMOTO BOMBA 096P001A";
   %DB78.DBX1.3 := "SELEC TAB MODO CAMPO BOMBA 096P001B";
   %DB78.DBX1.4 := "SELEC TAB MODO CCM BOMBA 096P001B";
   %DB78.DBX1.5 := "SELEC TAB MODO REMOTO BOMBA 096P001B";
   %DB78.DBX0.0 := "PARO EMERGENCIA TAB AGUA SERVICIO LOCAL";
   %DB78.DBX0.1 := "FALLA BREAKER TOTALIZADOR";
   %DB78.DBX0.2 := "FALLA BREAKER BOMBA 096P001A";
   %DB78.DBX0.3 := "FALLA BREAKER BOMBA 096P001B";
   %DB78.DBX0.4 := "FALLA BREAKER BOMBA 096P001C";
   %DB78.DBX0.5 := "FALLA BREAKER BOMBA 096P001D";
   %DB78.DBX0.6 := "FALLA BREAKER BOMBA 096P001E";
   %DB78.DBX0.7 := "FALLA BREAKER BOMBA 096P001F";
   %DB78.DBX3.0 := "SELEC TAB MODO REMOTO BOMBA 096P001E";
   %DB78.DBX3.1 := "SELEC TAB MODO CAMPO BOMBA 096P001F";
   %DB78.DBX3.2 := "SELEC TAB MODO CCM BOMBA 096P001F";
   %DB78.DBX3.3 := "SELEC TAB MODO REMOTO BOMBA 096P001F";
   %DB78.DBX2.0 := "SELEC TAB MODO CAMPO BOMBA 096P001C";
   %DB78.DBX2.1 := "SELEC TAB MODO CCM BOMBA 096P001C";
   %DB78.DBX2.2 := "SELEC TAB MODO REMOTO BOMBA 096P001C";
   %DB78.DBX2.3 := "SELEC TAB MODO CAMPO BOMBA 096P001D";
   %DB78.DBX2.4 := "SELEC TAB MODO CCM BOMBA 096P001D";
   %DB78.DBX2.5 := "SELEC TAB MODO REMOTO BOMBA 096P001D";
   %DB78.DBX2.6 := "SELEC TAB MODO CAMPO BOMBA 096P001E";
   %DB78.DBX2.7 := "SELEC TAB MODO CCM BOMBA 096P001E";
   %DB78.DBX5.0 := "PERMISO DE ARRANQUE";
   %DB78.DBX5.1 := "Tag_1";
   %DB78.DBX4.0 := "SWITCH DE BAJA PRESION AGUA DE SERVICIO";
   %DB78.DBX4.1 := "SWITCH DE FLUJO AGUA DE SERVICIO";
   %DB78.DBX4.2 := "PARO EMERGENCIA 096P001A CAMPO";
   %DB78.DBX4.3 := "PARO EMERGENCIA 096P001B CAMPO";
   %DB78.DBX4.4 := "PARO EMERGENCIA 096P001C CAMPO";
   %DB78.DBX4.5 := "PARO EMERGENCIA 096P001D CAMPO";
   %DB78.DBX4.6 := "PARO EMERGENCIA 096P001E CAMPO";
   %DB78.DBX4.7 := "PARO EMERGENCIA 096P001F CAMPO";
END_REGION

REGION Network 3: SALIDAS DIGITALES
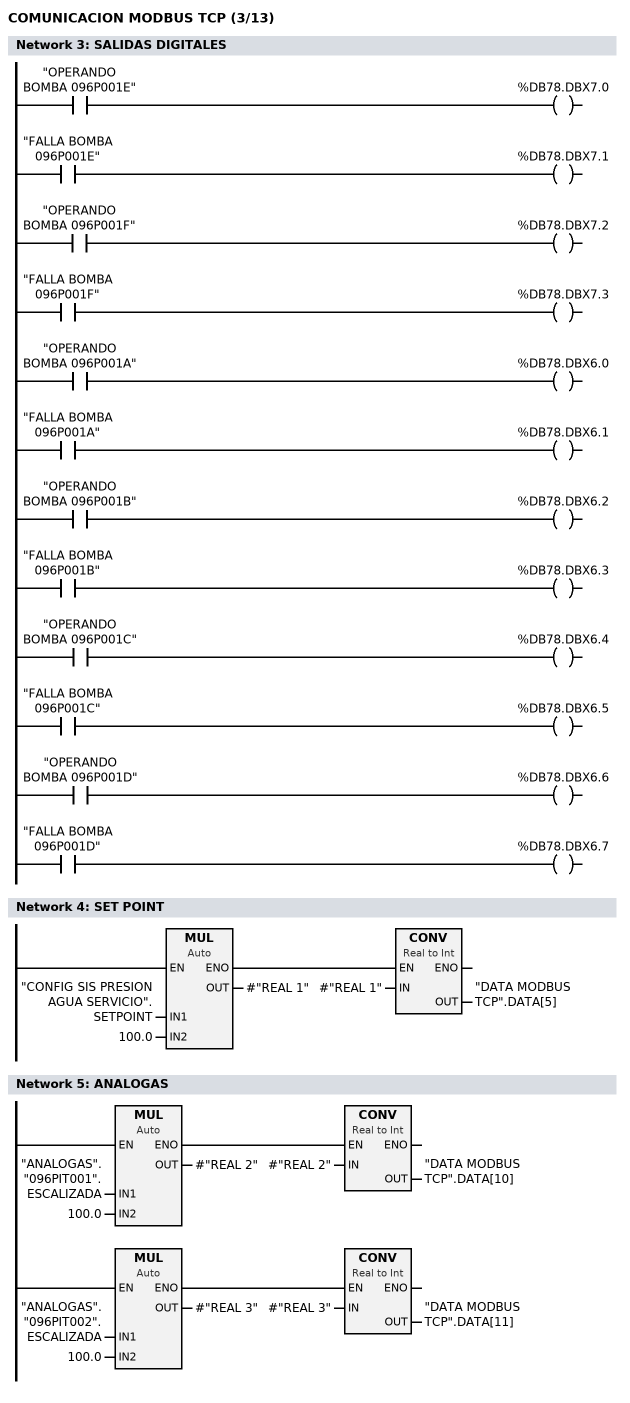
   RUNG wire#powerrail
      Contact( "OPERANDO BOMBA 096P001E" )
      Coil( %DB78.DBX7.0 )
   END_RUNG
   RUNG wire#powerrail
      Contact( "FALLA BOMBA 096P001E" )
      Coil( %DB78.DBX7.1 )
   END_RUNG
   RUNG wire#powerrail
      Contact( "OPERANDO BOMBA 096P001F" )
      Coil( %DB78.DBX7.2 )
   END_RUNG
   RUNG wire#powerrail
      Contact( "FALLA BOMBA 096P001F" )
      Coil( %DB78.DBX7.3 )
   END_RUNG
   RUNG wire#powerrail
      Contact( "OPERANDO BOMBA 096P001A" )
      Coil( %DB78.DBX6.0 )
   END_RUNG
   RUNG wire#powerrail
      Contact( "FALLA BOMBA 096P001A" )
      Coil( %DB78.DBX6.1 )
   END_RUNG
   RUNG wire#powerrail
      Contact( "OPERANDO BOMBA 096P001B" )
      Coil( %DB78.DBX6.2 )
   END_RUNG
   RUNG wire#powerrail
      Contact( "FALLA BOMBA 096P001B" )
      Coil( %DB78.DBX6.3 )
   END_RUNG
   RUNG wire#powerrail
      Contact( "OPERANDO BOMBA 096P001C" )
      Coil( %DB78.DBX6.4 )
   END_RUNG
   RUNG wire#powerrail
      Contact( "FALLA BOMBA 096P001C" )
      Coil( %DB78.DBX6.5 )
   END_RUNG
   RUNG wire#powerrail
      Contact( "OPERANDO BOMBA 096P001D" )
      Coil( %DB78.DBX6.6 )
   END_RUNG
   RUNG wire#powerrail
      Contact( "FALLA BOMBA 096P001D" )
      Coil( %DB78.DBX6.7 )
   END_RUNG
   // the same network as SCL:
   %DB78.DBX7.0 := "OPERANDO BOMBA 096P001E";
   %DB78.DBX7.1 := "FALLA BOMBA 096P001E";
   %DB78.DBX7.2 := "OPERANDO BOMBA 096P001F";
   %DB78.DBX7.3 := "FALLA BOMBA 096P001F";
   %DB78.DBX6.0 := "OPERANDO BOMBA 096P001A";
   %DB78.DBX6.1 := "FALLA BOMBA 096P001A";
   %DB78.DBX6.2 := "OPERANDO BOMBA 096P001B";
   %DB78.DBX6.3 := "FALLA BOMBA 096P001B";
   %DB78.DBX6.4 := "OPERANDO BOMBA 096P001C";
   %DB78.DBX6.5 := "FALLA BOMBA 096P001C";
   %DB78.DBX6.6 := "OPERANDO BOMBA 096P001D";
   %DB78.DBX6.7 := "FALLA BOMBA 096P001D";
END_REGION

REGION Network 4: SET POINT
   RUNG wire#powerrail
      Mul(in1 := "CONFIG SIS PRESION AGUA SERVICIO".SETPOINT, in2 := 100.0, out => #"REAL 1")
      { S7_Templates := "[SrcType := Real, DestType := Int]" } Convert(in := #"REAL 1", out => "DATA MODBUS TCP".DATA[5])
   END_RUNG
   // the same network as SCL:
   #"REAL 1" := "CONFIG SIS PRESION AGUA SERVICIO".SETPOINT * 100.0;
   "DATA MODBUS TCP".DATA[5] := REAL_TO_INT(#"REAL 1");
END_REGION

REGION Network 5: ANALOGAS
   RUNG wire#powerrail
      Mul(in1 := "ANALOGAS"."096PIT001".ESCALIZADA, in2 := 100.0, out => #"REAL 2")
      { S7_Templates := "[SrcType := Real, DestType := Int]" } Convert(in := #"REAL 2", out => "DATA MODBUS TCP".DATA[10])
   END_RUNG
   RUNG wire#powerrail
      Mul(in1 := "ANALOGAS"."096PIT002".ESCALIZADA, in2 := 100.0, out => #"REAL 3")
      { S7_Templates := "[SrcType := Real, DestType := Int]" } Convert(in := #"REAL 3", out => "DATA MODBUS TCP".DATA[11])
   END_RUNG
   // the same network as SCL:
   #"REAL 2" := "ANALOGAS"."096PIT001".ESCALIZADA * 100.0;
   "DATA MODBUS TCP".DATA[10] := REAL_TO_INT(#"REAL 2");
   #"REAL 3" := "ANALOGAS"."096PIT002".ESCALIZADA * 100.0;
   "DATA MODBUS TCP".DATA[11] := REAL_TO_INT(#"REAL 3");
END_REGION

REGION Network 6: VFD1
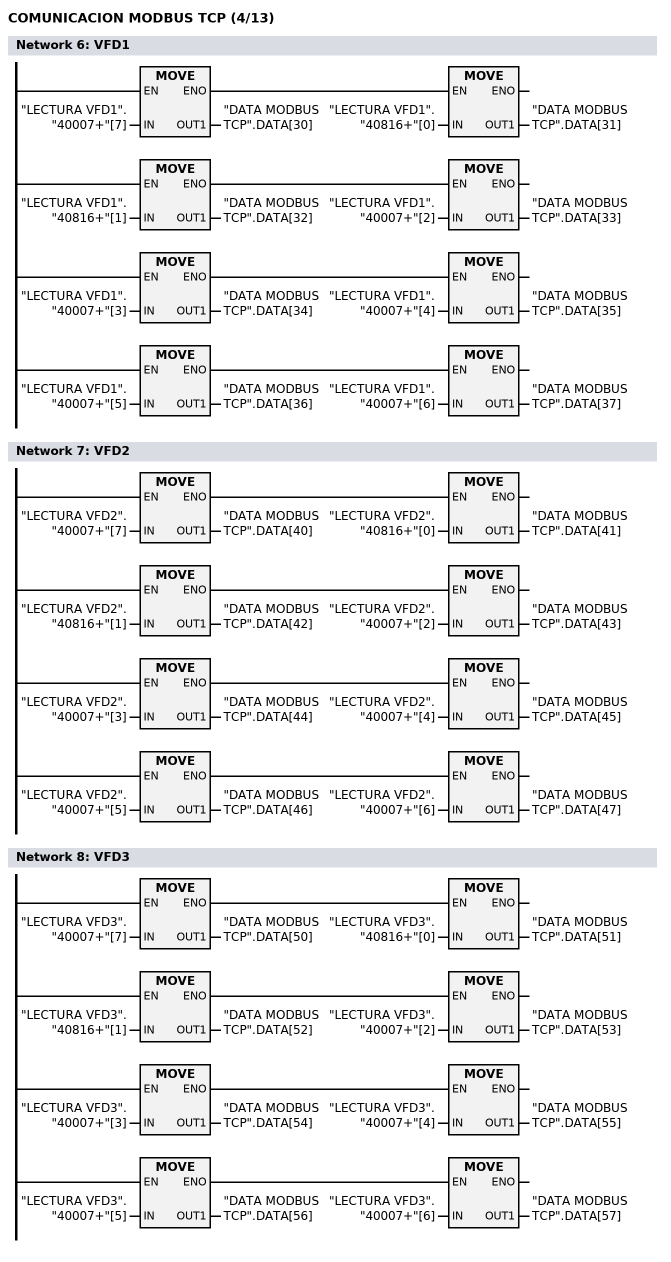
   RUNG wire#powerrail
      Move(in := "LECTURA VFD1"."40007+"[7], out1 => "DATA MODBUS TCP".DATA[30])
      Move(in := "LECTURA VFD1"."40816+"[0], out1 => "DATA MODBUS TCP".DATA[31])
   END_RUNG
   RUNG wire#powerrail
      Move(in := "LECTURA VFD1"."40816+"[1], out1 => "DATA MODBUS TCP".DATA[32])
      Move(in := "LECTURA VFD1"."40007+"[2], out1 => "DATA MODBUS TCP".DATA[33])
   END_RUNG
   RUNG wire#powerrail
      Move(in := "LECTURA VFD1"."40007+"[3], out1 => "DATA MODBUS TCP".DATA[34])
      Move(in := "LECTURA VFD1"."40007+"[4], out1 => "DATA MODBUS TCP".DATA[35])
   END_RUNG
   RUNG wire#powerrail
      Move(in := "LECTURA VFD1"."40007+"[5], out1 => "DATA MODBUS TCP".DATA[36])
      Move(in := "LECTURA VFD1"."40007+"[6], out1 => "DATA MODBUS TCP".DATA[37])
   END_RUNG
   // the same network as SCL:
   "DATA MODBUS TCP".DATA[30] := "LECTURA VFD1"."40007+"[7];
   "DATA MODBUS TCP".DATA[31] := "LECTURA VFD1"."40816+"[0];
   "DATA MODBUS TCP".DATA[32] := "LECTURA VFD1"."40816+"[1];
   "DATA MODBUS TCP".DATA[33] := "LECTURA VFD1"."40007+"[2];
   "DATA MODBUS TCP".DATA[34] := "LECTURA VFD1"."40007+"[3];
   "DATA MODBUS TCP".DATA[35] := "LECTURA VFD1"."40007+"[4];
   "DATA MODBUS TCP".DATA[36] := "LECTURA VFD1"."40007+"[5];
   "DATA MODBUS TCP".DATA[37] := "LECTURA VFD1"."40007+"[6];
END_REGION

REGION Network 7: VFD2
   RUNG wire#powerrail
      Move(in := "LECTURA VFD2"."40007+"[7], out1 => "DATA MODBUS TCP".DATA[40])
      Move(in := "LECTURA VFD2"."40816+"[0], out1 => "DATA MODBUS TCP".DATA[41])
   END_RUNG
   RUNG wire#powerrail
      Move(in := "LECTURA VFD2"."40816+"[1], out1 => "DATA MODBUS TCP".DATA[42])
      Move(in := "LECTURA VFD2"."40007+"[2], out1 => "DATA MODBUS TCP".DATA[43])
   END_RUNG
   RUNG wire#powerrail
      Move(in := "LECTURA VFD2"."40007+"[3], out1 => "DATA MODBUS TCP".DATA[44])
      Move(in := "LECTURA VFD2"."40007+"[4], out1 => "DATA MODBUS TCP".DATA[45])
   END_RUNG
   RUNG wire#powerrail
      Move(in := "LECTURA VFD2"."40007+"[5], out1 => "DATA MODBUS TCP".DATA[46])
      Move(in := "LECTURA VFD2"."40007+"[6], out1 => "DATA MODBUS TCP".DATA[47])
   END_RUNG
   // the same network as SCL:
   "DATA MODBUS TCP".DATA[40] := "LECTURA VFD2"."40007+"[7];
   "DATA MODBUS TCP".DATA[41] := "LECTURA VFD2"."40816+"[0];
   "DATA MODBUS TCP".DATA[42] := "LECTURA VFD2"."40816+"[1];
   "DATA MODBUS TCP".DATA[43] := "LECTURA VFD2"."40007+"[2];
   "DATA MODBUS TCP".DATA[44] := "LECTURA VFD2"."40007+"[3];
   "DATA MODBUS TCP".DATA[45] := "LECTURA VFD2"."40007+"[4];
   "DATA MODBUS TCP".DATA[46] := "LECTURA VFD2"."40007+"[5];
   "DATA MODBUS TCP".DATA[47] := "LECTURA VFD2"."40007+"[6];
END_REGION

REGION Network 8: VFD3
   RUNG wire#powerrail
      Move(in := "LECTURA VFD3"."40007+"[7], out1 => "DATA MODBUS TCP".DATA[50])
      Move(in := "LECTURA VFD3"."40816+"[0], out1 => "DATA MODBUS TCP".DATA[51])
   END_RUNG
   RUNG wire#powerrail
      Move(in := "LECTURA VFD3"."40816+"[1], out1 => "DATA MODBUS TCP".DATA[52])
      Move(in := "LECTURA VFD3"."40007+"[2], out1 => "DATA MODBUS TCP".DATA[53])
   END_RUNG
   RUNG wire#powerrail
      Move(in := "LECTURA VFD3"."40007+"[3], out1 => "DATA MODBUS TCP".DATA[54])
      Move(in := "LECTURA VFD3"."40007+"[4], out1 => "DATA MODBUS TCP".DATA[55])
   END_RUNG
   RUNG wire#powerrail
      Move(in := "LECTURA VFD3"."40007+"[5], out1 => "DATA MODBUS TCP".DATA[56])
      Move(in := "LECTURA VFD3"."40007+"[6], out1 => "DATA MODBUS TCP".DATA[57])
   END_RUNG
   // the same network as SCL:
   "DATA MODBUS TCP".DATA[50] := "LECTURA VFD3"."40007+"[7];
   "DATA MODBUS TCP".DATA[51] := "LECTURA VFD3"."40816+"[0];
   "DATA MODBUS TCP".DATA[52] := "LECTURA VFD3"."40816+"[1];
   "DATA MODBUS TCP".DATA[53] := "LECTURA VFD3"."40007+"[2];
   "DATA MODBUS TCP".DATA[54] := "LECTURA VFD3"."40007+"[3];
   "DATA MODBUS TCP".DATA[55] := "LECTURA VFD3"."40007+"[4];
   "DATA MODBUS TCP".DATA[56] := "LECTURA VFD3"."40007+"[5];
   "DATA MODBUS TCP".DATA[57] := "LECTURA VFD3"."40007+"[6];
END_REGION

REGION Network 9: VFD4
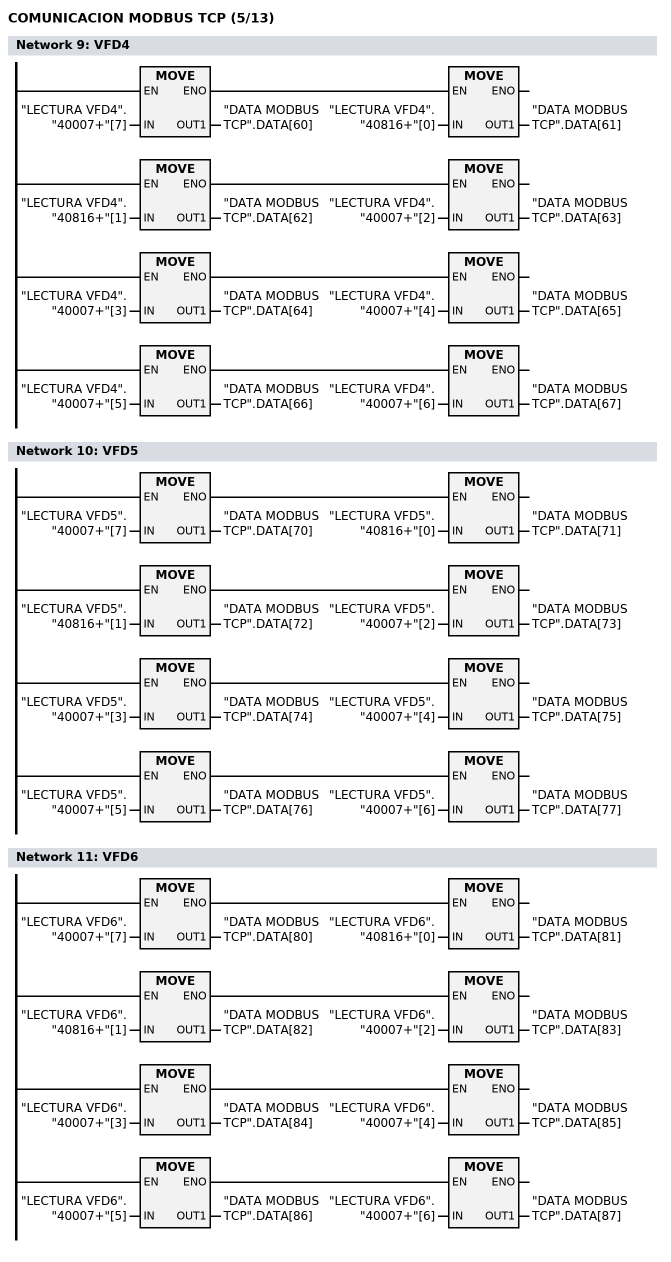
   RUNG wire#powerrail
      Move(in := "LECTURA VFD4"."40007+"[7], out1 => "DATA MODBUS TCP".DATA[60])
      Move(in := "LECTURA VFD4"."40816+"[0], out1 => "DATA MODBUS TCP".DATA[61])
   END_RUNG
   RUNG wire#powerrail
      Move(in := "LECTURA VFD4"."40816+"[1], out1 => "DATA MODBUS TCP".DATA[62])
      Move(in := "LECTURA VFD4"."40007+"[2], out1 => "DATA MODBUS TCP".DATA[63])
   END_RUNG
   RUNG wire#powerrail
      Move(in := "LECTURA VFD4"."40007+"[3], out1 => "DATA MODBUS TCP".DATA[64])
      Move(in := "LECTURA VFD4"."40007+"[4], out1 => "DATA MODBUS TCP".DATA[65])
   END_RUNG
   RUNG wire#powerrail
      Move(in := "LECTURA VFD4"."40007+"[5], out1 => "DATA MODBUS TCP".DATA[66])
      Move(in := "LECTURA VFD4"."40007+"[6], out1 => "DATA MODBUS TCP".DATA[67])
   END_RUNG
   // the same network as SCL:
   "DATA MODBUS TCP".DATA[60] := "LECTURA VFD4"."40007+"[7];
   "DATA MODBUS TCP".DATA[61] := "LECTURA VFD4"."40816+"[0];
   "DATA MODBUS TCP".DATA[62] := "LECTURA VFD4"."40816+"[1];
   "DATA MODBUS TCP".DATA[63] := "LECTURA VFD4"."40007+"[2];
   "DATA MODBUS TCP".DATA[64] := "LECTURA VFD4"."40007+"[3];
   "DATA MODBUS TCP".DATA[65] := "LECTURA VFD4"."40007+"[4];
   "DATA MODBUS TCP".DATA[66] := "LECTURA VFD4"."40007+"[5];
   "DATA MODBUS TCP".DATA[67] := "LECTURA VFD4"."40007+"[6];
END_REGION

REGION Network 10: VFD5
   RUNG wire#powerrail
      Move(in := "LECTURA VFD5"."40007+"[7], out1 => "DATA MODBUS TCP".DATA[70])
      Move(in := "LECTURA VFD5"."40816+"[0], out1 => "DATA MODBUS TCP".DATA[71])
   END_RUNG
   RUNG wire#powerrail
      Move(in := "LECTURA VFD5"."40816+"[1], out1 => "DATA MODBUS TCP".DATA[72])
      Move(in := "LECTURA VFD5"."40007+"[2], out1 => "DATA MODBUS TCP".DATA[73])
   END_RUNG
   RUNG wire#powerrail
      Move(in := "LECTURA VFD5"."40007+"[3], out1 => "DATA MODBUS TCP".DATA[74])
      Move(in := "LECTURA VFD5"."40007+"[4], out1 => "DATA MODBUS TCP".DATA[75])
   END_RUNG
   RUNG wire#powerrail
      Move(in := "LECTURA VFD5"."40007+"[5], out1 => "DATA MODBUS TCP".DATA[76])
      Move(in := "LECTURA VFD5"."40007+"[6], out1 => "DATA MODBUS TCP".DATA[77])
   END_RUNG
   // the same network as SCL:
   "DATA MODBUS TCP".DATA[70] := "LECTURA VFD5"."40007+"[7];
   "DATA MODBUS TCP".DATA[71] := "LECTURA VFD5"."40816+"[0];
   "DATA MODBUS TCP".DATA[72] := "LECTURA VFD5"."40816+"[1];
   "DATA MODBUS TCP".DATA[73] := "LECTURA VFD5"."40007+"[2];
   "DATA MODBUS TCP".DATA[74] := "LECTURA VFD5"."40007+"[3];
   "DATA MODBUS TCP".DATA[75] := "LECTURA VFD5"."40007+"[4];
   "DATA MODBUS TCP".DATA[76] := "LECTURA VFD5"."40007+"[5];
   "DATA MODBUS TCP".DATA[77] := "LECTURA VFD5"."40007+"[6];
END_REGION

REGION Network 11: VFD6
   RUNG wire#powerrail
      Move(in := "LECTURA VFD6"."40007+"[7], out1 => "DATA MODBUS TCP".DATA[80])
      Move(in := "LECTURA VFD6"."40816+"[0], out1 => "DATA MODBUS TCP".DATA[81])
   END_RUNG
   RUNG wire#powerrail
      Move(in := "LECTURA VFD6"."40816+"[1], out1 => "DATA MODBUS TCP".DATA[82])
      Move(in := "LECTURA VFD6"."40007+"[2], out1 => "DATA MODBUS TCP".DATA[83])
   END_RUNG
   RUNG wire#powerrail
      Move(in := "LECTURA VFD6"."40007+"[3], out1 => "DATA MODBUS TCP".DATA[84])
      Move(in := "LECTURA VFD6"."40007+"[4], out1 => "DATA MODBUS TCP".DATA[85])
   END_RUNG
   RUNG wire#powerrail
      Move(in := "LECTURA VFD6"."40007+"[5], out1 => "DATA MODBUS TCP".DATA[86])
      Move(in := "LECTURA VFD6"."40007+"[6], out1 => "DATA MODBUS TCP".DATA[87])
   END_RUNG
   // the same network as SCL:
   "DATA MODBUS TCP".DATA[80] := "LECTURA VFD6"."40007+"[7];
   "DATA MODBUS TCP".DATA[81] := "LECTURA VFD6"."40816+"[0];
   "DATA MODBUS TCP".DATA[82] := "LECTURA VFD6"."40816+"[1];
   "DATA MODBUS TCP".DATA[83] := "LECTURA VFD6"."40007+"[2];
   "DATA MODBUS TCP".DATA[84] := "LECTURA VFD6"."40007+"[3];
   "DATA MODBUS TCP".DATA[85] := "LECTURA VFD6"."40007+"[4];
   "DATA MODBUS TCP".DATA[86] := "LECTURA VFD6"."40007+"[5];
   "DATA MODBUS TCP".DATA[87] := "LECTURA VFD6"."40007+"[6];
END_REGION

REGION Network 12: ORDEN DE CAMBIO DE MODO BOMBA A
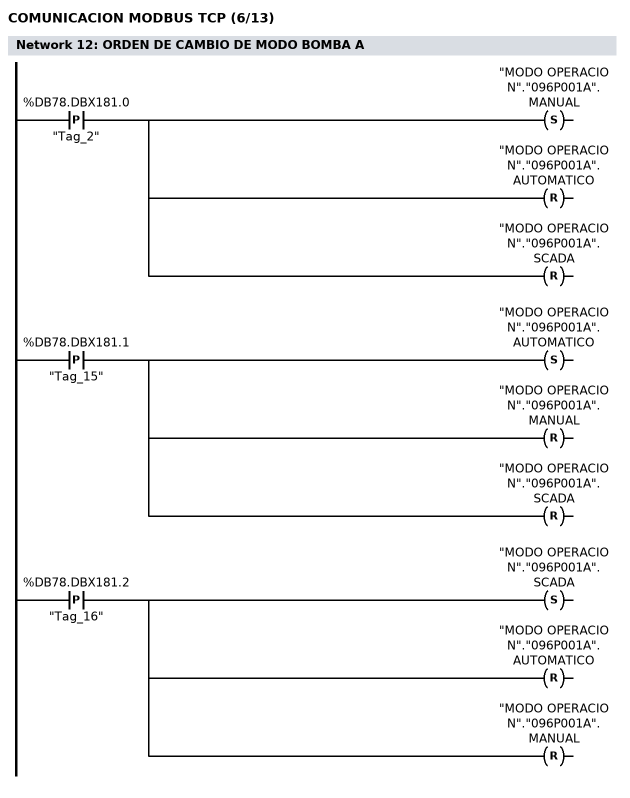
   RUNG wire#powerrail
      P_Contact(operand := %DB78.DBX181.0, bit := "Tag_2")
      wire#w1
      S_Coil( "MODO OPERACION"."096P001A".MANUAL )
   END_RUNG
   RUNG wire#w1
      R_Coil( "MODO OPERACION"."096P001A".AUTOMATICO )
   END_RUNG
   RUNG wire#w1
      R_Coil( "MODO OPERACION"."096P001A".SCADA )
   END_RUNG
   RUNG wire#powerrail
      P_Contact(operand := %DB78.DBX181.1, bit := "Tag_15")
      wire#w2
      S_Coil( "MODO OPERACION"."096P001A".AUTOMATICO )
   END_RUNG
   RUNG wire#w2
      R_Coil( "MODO OPERACION"."096P001A".MANUAL )
   END_RUNG
   RUNG wire#w2
      R_Coil( "MODO OPERACION"."096P001A".SCADA )
   END_RUNG
   RUNG wire#powerrail
      P_Contact(operand := %DB78.DBX181.2, bit := "Tag_16")
      wire#w3
      S_Coil( "MODO OPERACION"."096P001A".SCADA )
   END_RUNG
   RUNG wire#w3
      R_Coil( "MODO OPERACION"."096P001A".AUTOMATICO )
   END_RUNG
   RUNG wire#w3
      R_Coil( "MODO OPERACION"."096P001A".MANUAL )
   END_RUNG
   // the same network as SCL:
   #_w1 := %DB78.DBX181.0 AND NOT "Tag_2";   // rising edge of %DB78.DBX181.0
   "Tag_2" := %DB78.DBX181.0;
   IF #_w1 THEN
       "MODO OPERACION"."096P001A".MANUAL := TRUE;
       "MODO OPERACION"."096P001A".AUTOMATICO := FALSE;
       "MODO OPERACION"."096P001A".SCADA := FALSE;
   END_IF;
   #_w2 := %DB78.DBX181.1 AND NOT "Tag_15";   // rising edge of %DB78.DBX181.1
   "Tag_15" := %DB78.DBX181.1;
   IF #_w2 THEN
       "MODO OPERACION"."096P001A".AUTOMATICO := TRUE;
       "MODO OPERACION"."096P001A".MANUAL := FALSE;
       "MODO OPERACION"."096P001A".SCADA := FALSE;
   END_IF;
   #_w3 := %DB78.DBX181.2 AND NOT "Tag_16";   // rising edge of %DB78.DBX181.2
   "Tag_16" := %DB78.DBX181.2;
   IF #_w3 THEN
       "MODO OPERACION"."096P001A".SCADA := TRUE;
       "MODO OPERACION"."096P001A".AUTOMATICO := FALSE;
       "MODO OPERACION"."096P001A".MANUAL := FALSE;
   END_IF;
END_REGION

REGION Network 13: ORDEN DE CAMBIO DE MODO BOMBA B
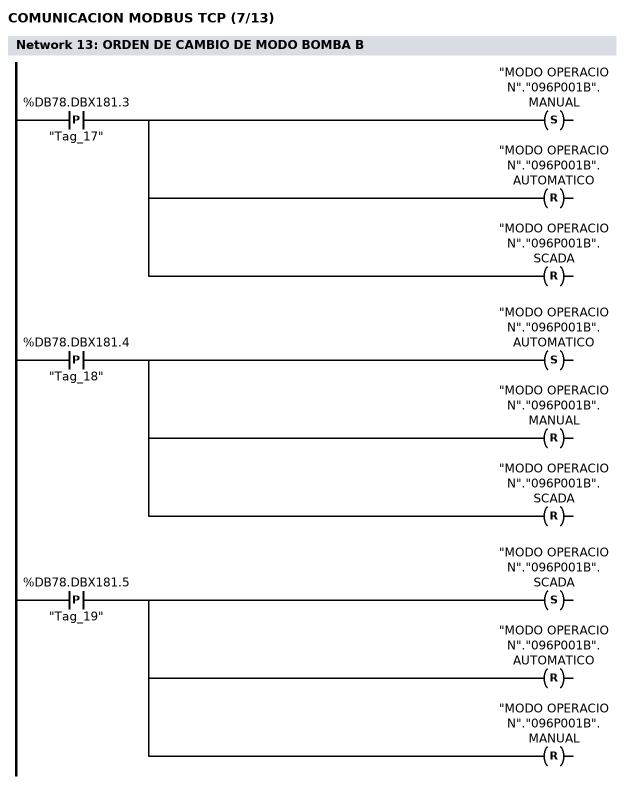
   RUNG wire#powerrail
      P_Contact(operand := %DB78.DBX181.3, bit := "Tag_17")
      wire#w1
      S_Coil( "MODO OPERACION"."096P001B".MANUAL )
   END_RUNG
   RUNG wire#w1
      R_Coil( "MODO OPERACION"."096P001B".AUTOMATICO )
   END_RUNG
   RUNG wire#w1
      R_Coil( "MODO OPERACION"."096P001B".SCADA )
   END_RUNG
   RUNG wire#powerrail
      P_Contact(operand := %DB78.DBX181.4, bit := "Tag_18")
      wire#w2
      S_Coil( "MODO OPERACION"."096P001B".AUTOMATICO )
   END_RUNG
   RUNG wire#w2
      R_Coil( "MODO OPERACION"."096P001B".MANUAL )
   END_RUNG
   RUNG wire#w2
      R_Coil( "MODO OPERACION"."096P001B".SCADA )
   END_RUNG
   RUNG wire#powerrail
      P_Contact(operand := %DB78.DBX181.5, bit := "Tag_19")
      wire#w3
      S_Coil( "MODO OPERACION"."096P001B".SCADA )
   END_RUNG
   RUNG wire#w3
      R_Coil( "MODO OPERACION"."096P001B".AUTOMATICO )
   END_RUNG
   RUNG wire#w3
      R_Coil( "MODO OPERACION"."096P001B".MANUAL )
   END_RUNG
   // the same network as SCL:
   #_w1 := %DB78.DBX181.3 AND NOT "Tag_17";   // rising edge of %DB78.DBX181.3
   "Tag_17" := %DB78.DBX181.3;
   IF #_w1 THEN
       "MODO OPERACION"."096P001B".MANUAL := TRUE;
       "MODO OPERACION"."096P001B".AUTOMATICO := FALSE;
       "MODO OPERACION"."096P001B".SCADA := FALSE;
   END_IF;
   #_w2 := %DB78.DBX181.4 AND NOT "Tag_18";   // rising edge of %DB78.DBX181.4
   "Tag_18" := %DB78.DBX181.4;
   IF #_w2 THEN
       "MODO OPERACION"."096P001B".AUTOMATICO := TRUE;
       "MODO OPERACION"."096P001B".MANUAL := FALSE;
       "MODO OPERACION"."096P001B".SCADA := FALSE;
   END_IF;
   #_w3 := %DB78.DBX181.5 AND NOT "Tag_19";   // rising edge of %DB78.DBX181.5
   "Tag_19" := %DB78.DBX181.5;
   IF #_w3 THEN
       "MODO OPERACION"."096P001B".SCADA := TRUE;
       "MODO OPERACION"."096P001B".AUTOMATICO := FALSE;
       "MODO OPERACION"."096P001B".MANUAL := FALSE;
   END_IF;
END_REGION

REGION Network 14: ORDEN DE CAMBIO DE MODO BOMBA C
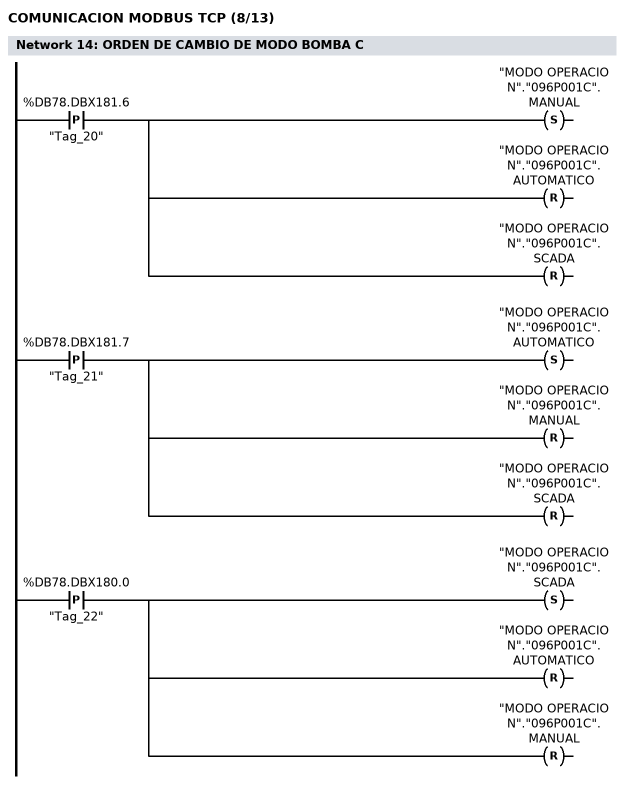
   RUNG wire#powerrail
      P_Contact(operand := %DB78.DBX181.6, bit := "Tag_20")
      wire#w1
      S_Coil( "MODO OPERACION"."096P001C".MANUAL )
   END_RUNG
   RUNG wire#w1
      R_Coil( "MODO OPERACION"."096P001C".AUTOMATICO )
   END_RUNG
   RUNG wire#w1
      R_Coil( "MODO OPERACION"."096P001C".SCADA )
   END_RUNG
   RUNG wire#powerrail
      P_Contact(operand := %DB78.DBX181.7, bit := "Tag_21")
      wire#w2
      S_Coil( "MODO OPERACION"."096P001C".AUTOMATICO )
   END_RUNG
   RUNG wire#w2
      R_Coil( "MODO OPERACION"."096P001C".MANUAL )
   END_RUNG
   RUNG wire#w2
      R_Coil( "MODO OPERACION"."096P001C".SCADA )
   END_RUNG
   RUNG wire#powerrail
      P_Contact(operand := %DB78.DBX180.0, bit := "Tag_22")
      wire#w3
      S_Coil( "MODO OPERACION"."096P001C".SCADA )
   END_RUNG
   RUNG wire#w3
      R_Coil( "MODO OPERACION"."096P001C".AUTOMATICO )
   END_RUNG
   RUNG wire#w3
      R_Coil( "MODO OPERACION"."096P001C".MANUAL )
   END_RUNG
   // the same network as SCL:
   #_w1 := %DB78.DBX181.6 AND NOT "Tag_20";   // rising edge of %DB78.DBX181.6
   "Tag_20" := %DB78.DBX181.6;
   IF #_w1 THEN
       "MODO OPERACION"."096P001C".MANUAL := TRUE;
       "MODO OPERACION"."096P001C".AUTOMATICO := FALSE;
       "MODO OPERACION"."096P001C".SCADA := FALSE;
   END_IF;
   #_w2 := %DB78.DBX181.7 AND NOT "Tag_21";   // rising edge of %DB78.DBX181.7
   "Tag_21" := %DB78.DBX181.7;
   IF #_w2 THEN
       "MODO OPERACION"."096P001C".AUTOMATICO := TRUE;
       "MODO OPERACION"."096P001C".MANUAL := FALSE;
       "MODO OPERACION"."096P001C".SCADA := FALSE;
   END_IF;
   #_w3 := %DB78.DBX180.0 AND NOT "Tag_22";   // rising edge of %DB78.DBX180.0
   "Tag_22" := %DB78.DBX180.0;
   IF #_w3 THEN
       "MODO OPERACION"."096P001C".SCADA := TRUE;
       "MODO OPERACION"."096P001C".AUTOMATICO := FALSE;
       "MODO OPERACION"."096P001C".MANUAL := FALSE;
   END_IF;
END_REGION

REGION Network 15: ORDEN DE CAMBIO DE MODO BOMBA D
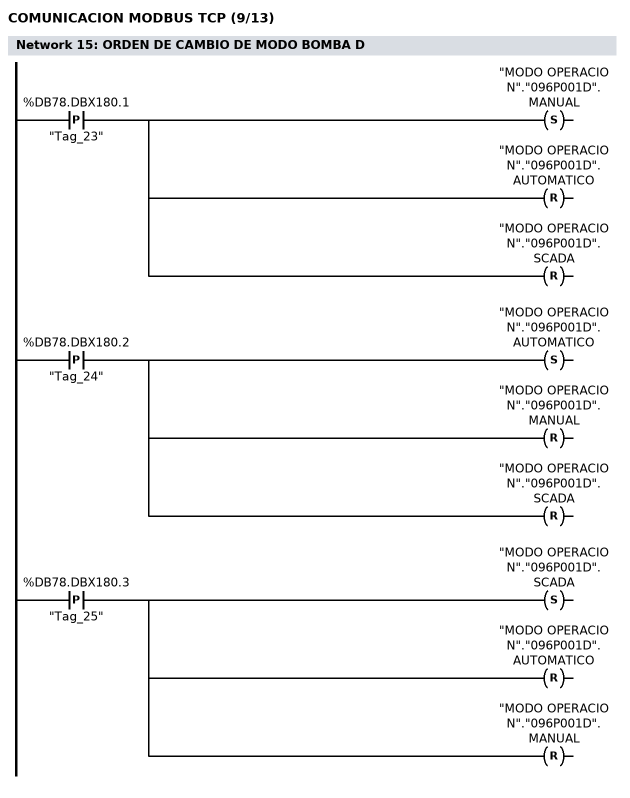
   RUNG wire#powerrail
      P_Contact(operand := %DB78.DBX180.1, bit := "Tag_23")
      wire#w1
      S_Coil( "MODO OPERACION"."096P001D".MANUAL )
   END_RUNG
   RUNG wire#w1
      R_Coil( "MODO OPERACION"."096P001D".AUTOMATICO )
   END_RUNG
   RUNG wire#w1
      R_Coil( "MODO OPERACION"."096P001D".SCADA )
   END_RUNG
   RUNG wire#powerrail
      P_Contact(operand := %DB78.DBX180.2, bit := "Tag_24")
      wire#w2
      S_Coil( "MODO OPERACION"."096P001D".AUTOMATICO )
   END_RUNG
   RUNG wire#w2
      R_Coil( "MODO OPERACION"."096P001D".MANUAL )
   END_RUNG
   RUNG wire#w2
      R_Coil( "MODO OPERACION"."096P001D".SCADA )
   END_RUNG
   RUNG wire#powerrail
      P_Contact(operand := %DB78.DBX180.3, bit := "Tag_25")
      wire#w3
      S_Coil( "MODO OPERACION"."096P001D".SCADA )
   END_RUNG
   RUNG wire#w3
      R_Coil( "MODO OPERACION"."096P001D".AUTOMATICO )
   END_RUNG
   RUNG wire#w3
      R_Coil( "MODO OPERACION"."096P001D".MANUAL )
   END_RUNG
   // the same network as SCL:
   #_w1 := %DB78.DBX180.1 AND NOT "Tag_23";   // rising edge of %DB78.DBX180.1
   "Tag_23" := %DB78.DBX180.1;
   IF #_w1 THEN
       "MODO OPERACION"."096P001D".MANUAL := TRUE;
       "MODO OPERACION"."096P001D".AUTOMATICO := FALSE;
       "MODO OPERACION"."096P001D".SCADA := FALSE;
   END_IF;
   #_w2 := %DB78.DBX180.2 AND NOT "Tag_24";   // rising edge of %DB78.DBX180.2
   "Tag_24" := %DB78.DBX180.2;
   IF #_w2 THEN
       "MODO OPERACION"."096P001D".AUTOMATICO := TRUE;
       "MODO OPERACION"."096P001D".MANUAL := FALSE;
       "MODO OPERACION"."096P001D".SCADA := FALSE;
   END_IF;
   #_w3 := %DB78.DBX180.3 AND NOT "Tag_25";   // rising edge of %DB78.DBX180.3
   "Tag_25" := %DB78.DBX180.3;
   IF #_w3 THEN
       "MODO OPERACION"."096P001D".SCADA := TRUE;
       "MODO OPERACION"."096P001D".AUTOMATICO := FALSE;
       "MODO OPERACION"."096P001D".MANUAL := FALSE;
   END_IF;
END_REGION

REGION Network 16: ORDEN DE CAMBIO DE MODO BOMBA E
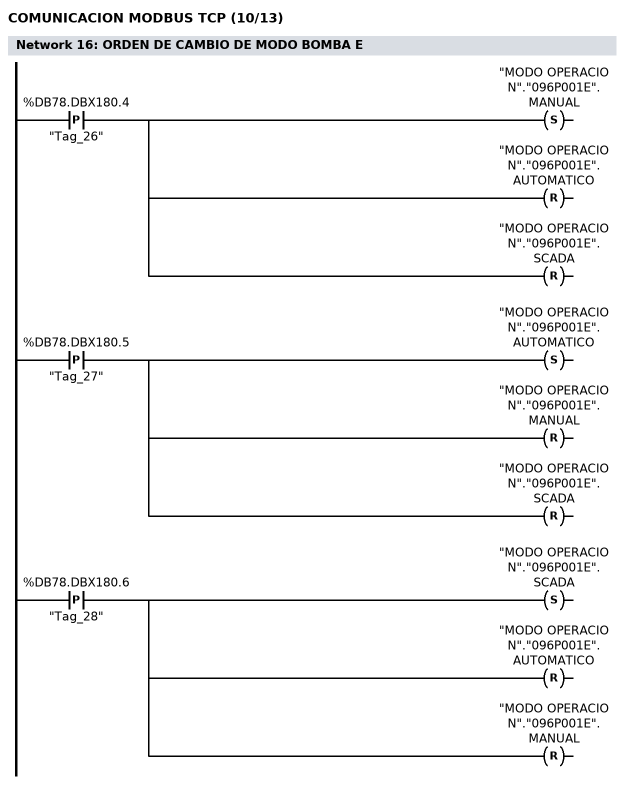
   RUNG wire#powerrail
      P_Contact(operand := %DB78.DBX180.4, bit := "Tag_26")
      wire#w1
      S_Coil( "MODO OPERACION"."096P001E".MANUAL )
   END_RUNG
   RUNG wire#w1
      R_Coil( "MODO OPERACION"."096P001E".AUTOMATICO )
   END_RUNG
   RUNG wire#w1
      R_Coil( "MODO OPERACION"."096P001E".SCADA )
   END_RUNG
   RUNG wire#powerrail
      P_Contact(operand := %DB78.DBX180.5, bit := "Tag_27")
      wire#w2
      S_Coil( "MODO OPERACION"."096P001E".AUTOMATICO )
   END_RUNG
   RUNG wire#w2
      R_Coil( "MODO OPERACION"."096P001E".MANUAL )
   END_RUNG
   RUNG wire#w2
      R_Coil( "MODO OPERACION"."096P001E".SCADA )
   END_RUNG
   RUNG wire#powerrail
      P_Contact(operand := %DB78.DBX180.6, bit := "Tag_28")
      wire#w3
      S_Coil( "MODO OPERACION"."096P001E".SCADA )
   END_RUNG
   RUNG wire#w3
      R_Coil( "MODO OPERACION"."096P001E".AUTOMATICO )
   END_RUNG
   RUNG wire#w3
      R_Coil( "MODO OPERACION"."096P001E".MANUAL )
   END_RUNG
   // the same network as SCL:
   #_w1 := %DB78.DBX180.4 AND NOT "Tag_26";   // rising edge of %DB78.DBX180.4
   "Tag_26" := %DB78.DBX180.4;
   IF #_w1 THEN
       "MODO OPERACION"."096P001E".MANUAL := TRUE;
       "MODO OPERACION"."096P001E".AUTOMATICO := FALSE;
       "MODO OPERACION"."096P001E".SCADA := FALSE;
   END_IF;
   #_w2 := %DB78.DBX180.5 AND NOT "Tag_27";   // rising edge of %DB78.DBX180.5
   "Tag_27" := %DB78.DBX180.5;
   IF #_w2 THEN
       "MODO OPERACION"."096P001E".AUTOMATICO := TRUE;
       "MODO OPERACION"."096P001E".MANUAL := FALSE;
       "MODO OPERACION"."096P001E".SCADA := FALSE;
   END_IF;
   #_w3 := %DB78.DBX180.6 AND NOT "Tag_28";   // rising edge of %DB78.DBX180.6
   "Tag_28" := %DB78.DBX180.6;
   IF #_w3 THEN
       "MODO OPERACION"."096P001E".SCADA := TRUE;
       "MODO OPERACION"."096P001E".AUTOMATICO := FALSE;
       "MODO OPERACION"."096P001E".MANUAL := FALSE;
   END_IF;
END_REGION

REGION Network 17: ORDEN DE CAMBIO DE MODO BOMBA F
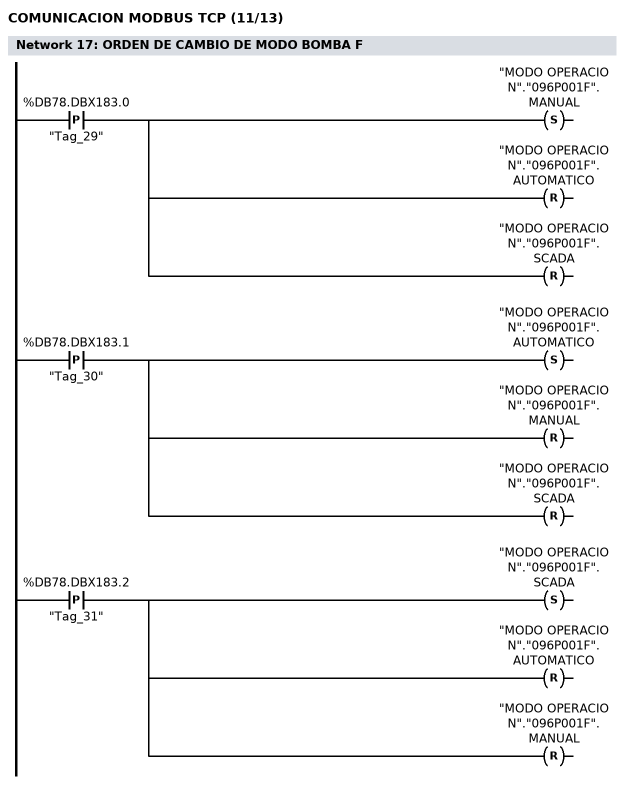
   RUNG wire#powerrail
      P_Contact(operand := %DB78.DBX183.0, bit := "Tag_29")
      wire#w1
      S_Coil( "MODO OPERACION"."096P001F".MANUAL )
   END_RUNG
   RUNG wire#w1
      R_Coil( "MODO OPERACION"."096P001F".AUTOMATICO )
   END_RUNG
   RUNG wire#w1
      R_Coil( "MODO OPERACION"."096P001F".SCADA )
   END_RUNG
   RUNG wire#powerrail
      P_Contact(operand := %DB78.DBX183.1, bit := "Tag_30")
      wire#w2
      S_Coil( "MODO OPERACION"."096P001F".AUTOMATICO )
   END_RUNG
   RUNG wire#w2
      R_Coil( "MODO OPERACION"."096P001F".MANUAL )
   END_RUNG
   RUNG wire#w2
      R_Coil( "MODO OPERACION"."096P001F".SCADA )
   END_RUNG
   RUNG wire#powerrail
      P_Contact(operand := %DB78.DBX183.2, bit := "Tag_31")
      wire#w3
      S_Coil( "MODO OPERACION"."096P001F".SCADA )
   END_RUNG
   RUNG wire#w3
      R_Coil( "MODO OPERACION"."096P001F".AUTOMATICO )
   END_RUNG
   RUNG wire#w3
      R_Coil( "MODO OPERACION"."096P001F".MANUAL )
   END_RUNG
   // the same network as SCL:
   #_w1 := %DB78.DBX183.0 AND NOT "Tag_29";   // rising edge of %DB78.DBX183.0
   "Tag_29" := %DB78.DBX183.0;
   IF #_w1 THEN
       "MODO OPERACION"."096P001F".MANUAL := TRUE;
       "MODO OPERACION"."096P001F".AUTOMATICO := FALSE;
       "MODO OPERACION"."096P001F".SCADA := FALSE;
   END_IF;
   #_w2 := %DB78.DBX183.1 AND NOT "Tag_30";   // rising edge of %DB78.DBX183.1
   "Tag_30" := %DB78.DBX183.1;
   IF #_w2 THEN
       "MODO OPERACION"."096P001F".AUTOMATICO := TRUE;
       "MODO OPERACION"."096P001F".MANUAL := FALSE;
       "MODO OPERACION"."096P001F".SCADA := FALSE;
   END_IF;
   #_w3 := %DB78.DBX183.2 AND NOT "Tag_31";   // rising edge of %DB78.DBX183.2
   "Tag_31" := %DB78.DBX183.2;
   IF #_w3 THEN
       "MODO OPERACION"."096P001F".SCADA := TRUE;
       "MODO OPERACION"."096P001F".AUTOMATICO := FALSE;
       "MODO OPERACION"."096P001F".MANUAL := FALSE;
   END_IF;
END_REGION

REGION Network 18: estados modos de operacion
